	//Kommunikationsfel
	fbKommTof : tof; 
	fbKommTon : ton;
		
	fb_CSP : Tc3_BA.FB_BA_Chrct02;
	
	sIP: STRING(255);
	sPort: STRING(255);
	sModbusID: STRING(255);
	sModbusLoop: STRING(255);
	
	sTemp: STRING(255);
END_VAR

//General
	offset := 0;
//Sekvens	
	bSekvensFlagga := oaksGVL.aBModbusSekvens[iModbusLoop] = UINT_TO_INT(nUnitID);
//Modbus konfiguering
	sIP := CONCAT (SIPAddr, '');
	sPort := CONCAT ('<br>Port: ', UINT_TO_STRING(nTCPPort)); 								
	sModbusID := CONCAT('<br>ID: ', UINT_TO_STRING(nUnitID));
	sModbusLoop := CONCAT('<br>Loop: ', INT_TO_STRING(iModbusLoop));
	
	sTemp := sIP;
	sTemp := CONCAT(sTemp, sPort);
	sTemp := CONCAT(sTemp, sModbusID);
	sTemp := CONCAT(sTemp, sModbusLoop);
	
	PV10 := sTemp;

///////////////		
//READ
///////////////		
	
	//Read Holding 0-8
	FB_MBReadRegs_ArrHolding1(
	sIPAddr:= sIpAddr, 
	nTCPPort:= INT_TO_UINT(nTCPPort), 
	nUnitID:= INT_TO_BYTE(nUnitID), 
	nQuantity:= 9, 
	nMBAddr:= 0 + offset, 
	cbLength:= SIZEOF(ArrHolding1), 
	pDestAddr:= ADR(ArrHolding1), 
	bExecute:= bSekvensFlagga, 
	tTimeout:= T#3S, 
	bBusy=> , 
	bError=> , 
	nErrId=> , 
	cbRead=> );
	
		//Values
		wActSetpoint := ArrHolding1[0]; //0
		wModeOut := ArrHolding1[1]; //1
		//ArrHolding1[2]; //2
		//ArrHolding1[3]; //3
		//ArrHolding1[4]; //4
		wRelPos := ArrHolding1[5]; //5
		//ArrHolding1[6]; //6
		wAbsVolume := ArrHolding1[7]; //7
		//ArrHolding1[8]; //8
							
		//Absolute Volume flow
		//Converter from m2 to l/s
		iTemp := WORD_TO_UINT(wAbsVolume);
		rTemp := UINT_TO_REAL(iTemp);
		PV1 := rTemp;
	
		//Relative Position
		iTemp := WORD_TO_UINT(wRelPos);
		rTemp := UINT_TO_REAL(iTemp);
		OP := rTemp / 100;
		
		//Actual damper-mode
		PV5 := wModeOut;
						
	//Read Holding 100-108
	FB_MBReadRegs_ArrHolding2(
	sIPAddr:= sIpAddr, 
	nTCPPort:= INT_TO_UINT(nTCPPort), 
	nUnitID:= INT_TO_BYTE(nUnitID), 
	nQuantity:= 9, 
	nMBAddr:= 100 + offset, 
	cbLength:= SIZEOF(ArrHolding2), 
	pDestAddr:= ADR(ArrHolding2), 
	bExecute:= bSekvensFlagga, 
	tTimeout:= T#3S, 
	bBusy=> , 
	bError=> , 
	nErrId=> , 
	cbRead=> );
	
		//Tilldela värden
		//ArrHolding2[100]; //100
		//ArrHolding2[101]; //101
		//ArrHolding2[102]; //102
		//ArrHolding2[103]; //103
		//ArrHolding2[104]; //104
		wAlarm := ArrHolding2[105]; //105
		//ArrHolding2[106]; //106
		//ArrHolding2[107]; //107
		//ArrHolding2[108]; //108
		
	
	//Read Holding 120-122
	FB_MBReadRegs_ArrHolding3(
	sIPAddr:= sIpAddr, 
	nTCPPort:= INT_TO_UINT(nTCPPort), 
	nUnitID:= INT_TO_BYTE(nUnitID), 
	nQuantity:= 3, 
	nMBAddr:= 120 + offset, 
	cbLength:= SIZEOF(ArrHolding3), 
	pDestAddr:= ADR(ArrHolding3), 
	bExecute:= bSekvensFlagga, 
	tTimeout:= T#3S, 
	bBusy=> , 
	bError=> , 
	nErrId=> , 
	cbRead=> );
	
		
		wMinVolume := ArrHolding3[120]; //120
		wMaxVolume := ArrHolding3[121]; //121		
		//ArrHolding3[122]; //122		
			
		//Setpoint Min-volume
		iTemp := WORD_TO_UINT(wMinVolume);
		PV6 := UINT_TO_REAL(iTemp);
						
		//Setpoint Max-volume
		iTemp := WORD_TO_UINT(wMaxVolume);
		PV7 := UINT_TO_REAL(iTemp);
		
	//Calculated setpoint
		fb_CSP(
			rX:= WORD_TO_REAL(wActSetpoint) / 100, 
			rX01:= 0, 
			rX02:= 100, 
			rY01:= PV6, 
			rY02:= PV7, 
			bLmt:= TRUE, 
			rY=> CSP, 
			bErr=> , 
			sErrDescr=> );

		
///////////////		
//WRITE
///////////////	
				
//Setpoint
	
	rTemp := LIMIT (0, rSetpoint, 100);
	wTemp := frealtoword(rTemp, 100);
		
	IF wTemp <> wActSetpoint AND bSekvensFlagga THEN
		FB_MBWriteSingleReg_Setpoint.bExecute := TRUE;
	ELSE
		FB_MBWriteSingleReg_Setpoint.bExecute := FALSE;
	END_IF
	
	//Write Setpoint
	FB_MBWriteSingleReg_Setpoint(
	sIPAddr:= sIpAddr, 
	nTCPPort:= INT_TO_UINT(nTCPPort), 
	nUnitID:= INT_TO_BYTE(nUnitID), 
	nMBAddr:= 0 + offset, 
	nValue:= wTemp, 
	bExecute:= , 
	tTimeout:= T#3S, 
	bBusy=> , 
	bError=> , 
	nErrId=> );
	
//Override
	
	iTemp := INT_TO_WORD(iMode);	

	IF wModeOut <> iTemp AND bSekvensFlagga THEN 
		FB_MBWriteSingleReg_Mode.bExecute := TRUE;
	ELSE 
		FB_MBWriteSingleReg_Mode.bExecute := FALSE;
	END_IF
	
	//Write Mode
	FB_MBWriteSingleReg_Mode(
	sIPAddr:= sIpAddr, 
	nTCPPort:= INT_TO_UINT(nTCPPort), 
	nUnitID:= INT_TO_BYTE(nUnitID), 
	nMBAddr:= 1 + offset, 
	nValue:= UINT_TO_WORD(iMode), 
	bExecute:= , 
	tTimeout:= T#3S, 
	bBusy=> , 
	bError=> , 
	nErrId=> );

//Read/write

//Min		
	fbWriteHoldingDoubleControlledMin(
	sIPAddr:= sIPAddr, 
	nTCPPort:= nTCPPort, 
	nUnitID:= UINT_TO_BYTE(nUnitID) , 
	nMBAddr:= 120+offset,
	bExecute:= bSekvensFlagga, 
	rScale:=1 , 
	rWrite:= SP1, 
	bBusy=> , 
	bError=> );
//Max
	fbWriteHoldingDoubleControlledMax(
	sIPAddr:= sIPAddr, 
	nTCPPort:= nTCPPort, 
	nUnitID:= UINT_TO_BYTE(nUnitID) , 
	nMBAddr:= 121+offset, 
	bExecute:=bSekvensFlagga , 
	rScale:=1 , 
	rWrite:=SP2 , 
	bBusy=> , 
	bError=> );
	
//Communication error
	fbKommTof(IN:=FB_MBReadRegs_ArrHolding1.bError , PT:=T#20S , Q=> , ET=> );
	fbKommTon(IN:=fbKommTof.Q , PT:=T#20M , Q=> , ET=> );
	FAULT :=fbKommTon.Q;
		
//Write busy	
	oaksgvl.aBModbusBusyFlagga[iModbusLoop,nUnitID] := FB_MBReadRegs_Arrholding1.bBusy OR FB_MBReadRegs_Arrholding2.bBusy OR FB_MBReadRegs_Arrholding3.bBusy OR FB_MBWriteSingleReg_Setpoint.bBusy OR FB_MBWriteSingleReg_Mode.bBusy;

END_FUNCTION_BLOCK

// oaksModbusLibrary/Frico/fbFricoSirE
// Modbusblock för frico sir e fläktluftvärmare fungerar bra men går att vidareutveckla med fler register
FUNCTION_BLOCK fbFricoSirE
VAR_INPUT
	sIPAddr : STRING := ''; 
	nTCPPort : UINT;
	nUnitID : UINT;
	iModbusLoop : INT :=1; //Modbusslinga
	M AT %M*  : BOOL;  //Reset summalarm~wp:
END_VAR
VAR_OUTPUT 
	V AT %M*  : BOOL;//Driftindikering~wp:[trendoptions]i:14400, t:1
	PV AT %M*  : REAL;//Temperatur~wp:[unit]°C[format]0.0[trendoptions]i:300
	PV1 AT %M*  : REAL;//Fläkthastighet~wp:[unit]%[format]0[trendoptions]i:300
	VALVE_OP AT %M*  : REAL;//Ventilläge~wp:[unit]%[format]0[trendoptions]i:300
	AL AT %M*  : BOOL; //Summalarm~wp:[trendoptions]i:300
	PV8 AT %M* : STRING;//Modbus konfiguering~wp:
	FAULT AT %M* : BOOL;//Kommunikationsfel~wp:[trendoptions]i:300
END_VAR
VAR
	sIP: STRING(255);
	sPort: STRING(255);
	sModbusID: STRING(255);
	sModbusLoop: STRING(255);
	sTemp : STRING(255);	


	//Kommunikationsfel
	fbKommTof : tof; 
	fbKommTon : ton;

	bSekvensFlagga : BOOL;	

	fbWriteToggle01,fbReadToggle : fbToggle;
	bExecute1,bExecute11,bExecute12 : BOOL;
	fbTemperature: FB_MBReadRegs;
	wWord :  ARRAY [1..9] OF WORD;
	wDaySetpointConfirmed,wNightSetpointConfirmed : WORD;
	
	
	
	fbWriteNight: FB_MBWriteSingleReg;
	wDaySetpoint : WORD;
	fbWriteToggle011 : fbToggle;
	
	fbWriteDay: FB_MBWriteSingleReg;
	wNightSetpoint : WORD;
	fbWriteToggle012 : fbToggle;
	
	
	wResetConfirmed : WORD;
		iTemp : INT;
	fbResetConfirmed : FB_MBReadRegs;
	fbWriteReset: FB_MBWriteSingleReg;
END_VAR
VAR_INPUT PERSISTENT
	SP AT %M*  : REAL := 18;  //Inställt börvärde~wp:[unit]°C[format]0.0[trendoptions]i:300
END_VAR

//Modbus konfiguering
	sIP := CONCAT (SIPAddr, '');
	sPort := CONCAT ('<br>Port: ', UINT_TO_STRING(nTCPPort)); 								
	sModbusID := CONCAT('<br>ID: ', UINT_TO_STRING(nUnitID));
	sModbusLoop := CONCAT('<br>Loop: ', INT_TO_STRING(iModbusLoop));	

	sTemp := sIP;
	sTemp := CONCAT(sTemp, sPort);
	sTemp := CONCAT(sTemp, sModbusID);
	sTemp := CONCAT(sTemp, sModbusLoop);
	
	PV8 := sTemp;

//Sekvens	
	bSekvensFlagga := oaksGVL.aBModbusSekvens[iModbusLoop] = UINT_TO_INT(nUnitID);

	fbTemperature(
	sIPAddr:= sIPAddr, 
	nTCPPort:= nTCPPort, 
	nUnitID:= UINT_TO_BYTE(nUnitID), 
	nQuantity:= 9, 
	nMBAddr:= 0, 
	cbLength:= SIZEOF(wWord), 
	pDestAddr:=ADR(wWord) , 
	bExecute:=bSekvensFlagga , 
	tTimeout:= T#5S, 
	bBusy=> , 
	bError=> , 
	nErrId=> , 
	cbRead=> );

	PV := fSignedConverter(WORD_TO_REAL(wWord[1])) * 0.1;
	PV1 := WORD_TO_REAL(wWord[3]);
	VALVE_OP :=  WORD_TO_REAL(wWord[4]);
	
	V := PV1 > 0.0;
	
	
	wDaySetpointConfirmed := wWord[8];
	wNightSetpointConfirmed := wWord[9];
	
	IF mBHyst(rProcessValue :=SP ,rSetPoint:=REAL_TO_WORD(wDaySetpointConfirmed) ,rDevLimit:=0.25) THEN
		wDaySetpoint := REAL_TO_WORD(SP);
		bExecute11 := TRUE;
	ELSE
		bExecute11 := FALSE;
	END_IF;
	
	fbWriteToggle011(bStart:=bExecute11 , bOutput=> );

	fbWriteDay(
	sIPAddr:= sIpAddr, 
	nTCPPort:= INT_TO_UINT(nTCPPort), 
	nUnitID:= INT_TO_BYTE(nUnitID), 
	nMBAddr:= 7, 
	nValue:= wDaySetpoint, 
	bExecute:= fbWriteToggle011.bOutput AND bSekvensFlagga, 
	tTimeout:=T#5S , 
	bBusy=> , 
	bError=> , 
	nErrId=> );
	
	IF mBHyst(rProcessValue :=SP ,rSetPoint:=REAL_TO_WORD(wNightSetpointConfirmed) ,rDevLimit:=0.25) THEN
		wNightSetpoint := REAL_TO_WORD(SP);
		bExecute12 := TRUE;
	ELSE
		bExecute12 := FALSE;
	END_IF;
	
	fbWriteToggle012(bStart:=bExecute12 , bOutput=> );

	fbWriteNight(
	sIPAddr:= sIpAddr, 
	nTCPPort:= INT_TO_UINT(nTCPPort), 
	nUnitID:= INT_TO_BYTE(nUnitID), 
	nMBAddr:= 8, 
	nValue:= wNightSetpoint, 
	bExecute:= fbWriteToggle012.bOutput AND bSekvensFlagga, 
	tTimeout:=T#5S , 
	bBusy=> , 
	bError=> , 
	nErrId=> );
(**** RESET START ****)
	IF M AND  wResetConfirmed = 0 THEN
		bExecute1 := TRUE;
	ELSE
		M := FALSE;
		bExecute1 := FALSE;
	END_IF;
	
	fbWriteToggle01(bStart:=bExecute1 , bOutput=> );

	fbWriteReset(
	sIPAddr:= sIpAddr, 
	nTCPPort:= INT_TO_UINT(nTCPPort), 
	nUnitID:= INT_TO_BYTE(nUnitID), 
	nMBAddr:= 99, 
	nValue:= 1, 
	bExecute:= fbWriteToggle01.bOutput AND bSekvensFlagga, 
	tTimeout:=T#1S , 
	bBusy=> , 
	bError=> , 
	nErrId=> );
	
	fbResetConfirmed(
	sIPAddr:= sIpAddr, 
	nTCPPort:= INT_TO_UINT(nTCPPort), 
	nUnitID:= INT_TO_BYTE(nUnitID), 
	nQuantity:= 1, 
	nMBAddr:= 99, 
	cbLength:= SIZEOF(wResetConfirmed), 
	pDestAddr:= ADR(wResetConfirmed), 
	bExecute:= bSekvensFlagga, 
	tTimeout:= T#1S, 
	bBusy=> , 
	bError=> , 
	nErrId=> , 
	cbRead=> );
	(**** RESET SLUT ****)
	
	//Communication error
	fbKommTof(IN:=fbTemperature.bError , PT:=T#20S , Q=> , ET=> );
	fbKommTon(IN:=fbKommTof.Q , PT:=T#20M , Q=> , ET=> );
	FAULT :=fbKommTon.Q;
		
//Write busy	
	oaksgvl.aBModbusBusyFlagga[iModbusLoop,nUnitID] := fbResetConfirmed.bBusy OR fbWriteReset.bBusy OR fbWriteNight.bBusy OR fbWriteDay.bBusy OR fbTemperature.bBusy;

METHOD PRIVATE mBHyst : BOOL
VAR_INPUT
	rProcessValue : REAL;
	rSetPoint : REAL; 
	rDevLimit : REAL;
END_VAR
VAR
END_VAR
	IF rProcessValue > (rSetPoint + rDevLimit)  THEN
		mBHyst := TRUE;
	ELSIF rProcessValue < (rSetPoint - rDevLimit)  THEN
		mBHyst := TRUE;
	ELSE	
		mBHyst := FALSE;
	END_IF;
END_METHOD

END_FUNCTION_BLOCK

// oaksModbusLibrary/Frico/fbFricoSirEOvride
// Modbusblock för frico sir e fläktluftvärmare fungerar bra men går att vidareutveckla med fler register
//2023-01-20 v2 Johan Stenström, Lagt till skicka utetemp., start/stopp, växling dag/natt

FUNCTION_BLOCK fbFricoSirEOvride
VAR_INPUT
	sIPAddr : STRING := ''; 
	nTCPPort : UINT := 502;
	nUnitID : UINT;
	iModbusLoop : INT := 1; //Modbusslinga
	iOnOff AT %M* : INT := 1; //Extern styrning till/från~wp:
	PV6 AT %M* : INT := 1; //Dag/Natt styrning börvärde, Dag=1, Natt=0~wp:
	ACK AT %M* : BOOL;  //Reset summalarm~wp:
END_VAR
VAR_OUTPUT 
	V AT %M*  : BOOL;//Driftindikering~wp:[trendoptions]i:14400, t:1
	CMD AT %M* : BOOL ; //Manöver~wp:[trendoptions]i:14400, t:1
	ROOM_PV AT %M*  : REAL;//Temperatur~wp:[unit]°C[format]0.0[trendoptions]i:300
	ROOM_CSP AT %M*  : REAL;//Aktuellt börvärde~wp:[unit]°C[format]0.0[trendoptions]i:300
	PV1 AT %M*  : REAL;//Fläkthastighet~wp:[unit]%[format]0[trendoptions]i:300
	VALVE_OP AT %M*  : REAL;//Ventilläge~wp:[unit]%[format]0[trendoptions]i:300
	AL AT %M*  : BOOL; //Summalarm~wp:[alarmoptions]p:2
	AL8 AT %M* : BOOL; //Utsignal handställd~wp:[alarmoptions]p:3
	PV8 AT %M* : STRING;//Modbus konfiguering~wp:
	FAULT AT %M* : BOOL;//Kommunikationsfel~wp:[trendoptions]i:300
END_VAR
VAR
	sIP: STRING(255);
	sPort: STRING(255);
	sModbusID: STRING(255);
	sModbusLoop: STRING(255);
	sTemp : STRING(255);	
	offset : WORD;
	fbAlarm1 : fbAlarm; // Larm handställning
//Kommunikationsfel
	fbKommTof : tof; 
	fbKommTon : ton;

	bSekvensFlagga : BOOL;	

	fbWriteToggle01 : fbToggle;
	bExecute1 : BOOL; 
	fbTemperature : FB_MBReadRegs;
	wWord :  ARRAY [1..12] OF WORD;
	wWordAlarm :  ARRAY [1..33] OF WORD;
	rOutDoorTempPointValueConfirmed : REAL;
	wSystemOnOffConfirmed, wWeekProgramConfirmed : WORD;
	wDaySetpointConfirmed, wNightSetpointConfirmed : WORD;
//OutDoorTemp	
	fbWriteOutDoorTemp : FB_MBWriteSingleReg;
	wOutDoorTempPointValue : WORD;
//SystemOnOff
	fbSystemOnOff : FB_MBWriteSingleReg;
	wSystemOnOff : WORD;
//WeekProgram
	fbWeekProgram : FB_MBWriteSingleReg;
	wWeekProgram : WORD;
//Setpoint Day	
	fbWriteDay : FB_MBWriteSingleReg;
	wDaySetpoint : WORD;
//Setpoint Night	
	fbWriteNight : FB_MBWriteSingleReg;
	wNightSetpoint : WORD;
//Alarm	
	fbAlarm : FB_MBReadRegs;
	wResetConfirmed : WORD;
//	iTemp : INT;
	fbResetConfirmed : FB_MBReadRegs;
	fbWriteReset : FB_MBWriteSingleReg;
	bAlarm01 : BOOL;
	bAlarm02 : BOOL; 
	bAlarm03 : BOOL; 
	bAlarm04 : BOOL; 
	bAlarm06 : BOOL;
	bAlarm07 : BOOL;
	bAlarm08 : BOOL; 
	bAlarm10 : BOOL; 
	bAlarm12 : BOOL; 
	bAlarm14 : BOOL;
	bAlarm21 : BOOL;
	bAlarm29 : BOOL;
	bAlarm30 : BOOL; 
	bAlarm31 : BOOL; 
	bAlarm32 : BOOL; 
	bAlarm33 : BOOL;  
	
END_VAR
VAR_INPUT PERSISTENT
	PV5 AT %M* : REAL;//Utetemperatur~wp:[unit]°C[format]0.0
	DAY_SP AT %M*  : REAL := 18;  //Börvärde dag~wp:[unit]°C[format]0.0[trendoptions]i:300
	NIGHT_SP AT %M*  : REAL := 16;  //Börvärde natt~wp:[unit]°C[format]0.0[trendoptions]i:300
	M AT %M* : BOOL; //Handställning~wp:
	MCMD AT %M* : BOOL; //Styrsignal handställning~wp:
END_VAR

//General
	offset := 0;
	fbAlarm1(bInput:=M, tAlarmDelay:= , bAutoReset:=TRUE , bAlarmOutput=>AL8 );
//Sekvens	
	bSekvensFlagga := oaksGVL.aBModbusSekvens[iModbusLoop] = UINT_TO_INT(nUnitID);
//Modbus konfiguering
	sIP := CONCAT (SIPAddr, '');
	sPort := CONCAT ('<br>Port: ', UINT_TO_STRING(nTCPPort)); 								
	sModbusID := CONCAT('<br>ID: ', UINT_TO_STRING(nUnitID));
	sModbusLoop := CONCAT('<br>Loop: ', INT_TO_STRING(iModbusLoop));	

	sTemp := sIP;
	sTemp := CONCAT(sTemp, sPort);
	sTemp := CONCAT(sTemp, sModbusID);
	sTemp := CONCAT(sTemp, sModbusLoop);
	
	PV8 := sTemp;
	
	IF PV6 > 0 THEN
		ROOM_CSP := DAY_SP;
	ELSE
		ROOM_CSP := NIGHT_SP;
	END_IF;

	fbTemperature(
	sIPAddr:= sIPAddr, 
	nTCPPort:= (nTCPPort), 
	nUnitID:= UINT_TO_BYTE(nUnitID), 
	nQuantity:= 10, 
	nMBAddr:= 0 + offset,
	cbLength:= SIZEOF(wWord), 
	pDestAddr:= ADR(wWord), 
	bExecute:= bSekvensFlagga, 
	tTimeout:= T#5S, 
	bBusy=> , 
	bError=> , 
	nErrId=> , 
	cbRead=> );

	ROOM_PV := fSignedConverter(WORD_TO_REAL(wWord[1])) * 0.1;
	rOutDoorTempPointValueConfirmed := fSignedConverter(WORD_TO_REAL(wWord[2]));
	PV1 := WORD_TO_REAL(wWord[3]);
	VALVE_OP :=  WORD_TO_REAL(wWord[4]);
	
	V := PV1 > 0.0;
	CMD := PV1 > 0.0;
	
	wSystemOnOffConfirmed := wWord[6];
	wWeekProgramConfirmed := wWord[7];
	wDaySetpointConfirmed := wWord[8];
	wNightSetpointConfirmed := wWord[9];
	
//OutDoorTemp	
	wOutDoorTempPointValue := fRealToWord(rReal:=PV5 , uiFaktor:= 10);
	
	fbWriteOutDoorTemp(
	sIPAddr:= sIpAddr, 
	nTCPPort:= INT_TO_UINT(nTCPPort), 
	nUnitID:= INT_TO_BYTE(nUnitID), 
	nMBAddr:= 1 + offset,
	nValue:= wOutDoorTempPointValue,
	bExecute:= bSekvensFlagga,
	tTimeout:=T#5S , 
	bBusy=> , 
	bError=> , 
	nErrId=> );	

//SystemOnOff	
	wSystemOnOff := INT_TO_WORD(iOnOff);
	
	IF M THEN
		IF (M AND MCMD) THEN
			wSystemOnOff := INT_TO_WORD(1);
		ELSE
			wSystemOnOff := INT_TO_WORD(0);
		END_IF
	ELSE
		wSystemOnOff := INT_TO_WORD(iOnOff);
	END_IF
	
	fbSystemOnOff(
	sIPAddr:= sIpAddr, 
	nTCPPort:= INT_TO_UINT(nTCPPort), 
	nUnitID:= INT_TO_BYTE(nUnitID), 
	nMBAddr:= 5 + offset, 
	nValue:= wSystemOnOff, 
	bExecute:= bSekvensFlagga,
	tTimeout:=T#5S , 
	bBusy=> , 
	bError=> , 
	nErrId=> );		
	
//WeekProgram
	IF PV6 > 0 THEN
		wWeekProgram := INT_TO_WORD(1);
	ELSE
		wWeekProgram := INT_TO_WORD(2);
	END_IF
	
	fbWeekProgram(
	sIPAddr:= sIpAddr, 
	nTCPPort:= INT_TO_UINT(nTCPPort), 
	nUnitID:= INT_TO_BYTE(nUnitID), 
	nMBAddr:= 6 + offset,
	nValue:= wWeekProgram, 
	bExecute:= bSekvensFlagga,
	tTimeout:=T#5S , 
	bBusy=> , 
	bError=> , 
	nErrId=> );		
	
//DaySetpoint
	wDaySetpoint := REAL_TO_WORD(DAY_SP);	

	fbWriteDay(
	sIPAddr:= sIpAddr, 
	nTCPPort:= INT_TO_UINT(nTCPPort), 
	nUnitID:= INT_TO_BYTE(nUnitID), 
	nMBAddr:= 7 + offset, 
	nValue:= wDaySetpoint, 
	bExecute:= bSekvensFlagga,
	tTimeout:=T#5S , 
	bBusy=> , 
	bError=> , 
	nErrId=> );
	
//WriteNight
	wNightSetpoint := REAL_TO_WORD(NIGHT_SP);

	fbWriteNight(
	sIPAddr:= sIpAddr, 
	nTCPPort:= INT_TO_UINT(nTCPPort), 
	nUnitID:= INT_TO_BYTE(nUnitID), 
	nMBAddr:= 8 + offset, 
	nValue:= wNightSetpoint, 
	bExecute:= bSekvensFlagga,
	tTimeout:=T#5S , 
	bBusy=> , 
	bError=> , 
	nErrId=> );
	
(**** ALARM ****)	
	bSekvensFlagga := oaksGVL.aBModbusSekvens[iModbusLoop] = UINT_TO_INT(nUnitID);

	fbAlarm(
	sIPAddr:= sIPAddr, 
	nTCPPort:= nTCPPort, 
	nUnitID:= UINT_TO_BYTE(nUnitID), 
	nQuantity:= 33, 
	nMBAddr:= 100 + offset, 
	cbLength:= SIZEOF(wWordAlarm), 
	pDestAddr:=ADR(wWordAlarm) , 
	bExecute:=bSekvensFlagga , 
	tTimeout:= T#5S, 
	bBusy=> , 
	bError=> , 
	nErrId=> , 
	cbRead=> );

	bAlarm01 := WORD_TO_BOOL(wWordAlarm[1]);
	bAlarm02 := WORD_TO_BOOL(wWordAlarm[2]);
	bAlarm03 := WORD_TO_BOOL(wWordAlarm[3]);
	bAlarm04 :=  WORD_TO_BOOL(wWordAlarm[4]);	
	bAlarm06 :=  WORD_TO_BOOL(wWordAlarm[6]);
	bAlarm07 :=  WORD_TO_BOOL(wWordAlarm[7]);
	bAlarm08 :=  WORD_TO_BOOL(wWordAlarm[8]);
	bAlarm10 :=  WORD_TO_BOOL(wWordAlarm[10]);
	bAlarm12 :=  WORD_TO_BOOL(wWordAlarm[12]);
	bAlarm14 :=  WORD_TO_BOOL(wWordAlarm[14]);
	bAlarm21 :=  WORD_TO_BOOL(wWordAlarm[21]);
	bAlarm29 :=  WORD_TO_BOOL(wWordAlarm[29]);
	bAlarm30 :=  WORD_TO_BOOL(wWordAlarm[30]);
	bAlarm31 :=  WORD_TO_BOOL(wWordAlarm[31]);
	bAlarm32 :=  WORD_TO_BOOL(wWordAlarm[32]);
	bAlarm33 :=  WORD_TO_BOOL(wWordAlarm[33]);
	
	IF bAlarm01 OR bAlarm02 OR bAlarm03 OR bAlarm04 OR bAlarm06 OR	bAlarm07 OR
		bAlarm08 OR bAlarm10 OR	bAlarm12 OR bAlarm14 OR bAlarm21 OR	bAlarm29 OR
		bAlarm30 OR bAlarm31 OR	bAlarm32 OR bAlarm33 = TRUE THEN
		AL := TRUE;
	ELSE
		AL := FALSE;
	END_IF;	
	
(**** RESET START ****)
	IF ACK AND  wResetConfirmed = 0 THEN
		bExecute1 := TRUE;
	ELSE
		ACK := FALSE;
		bExecute1 := FALSE;
	END_IF;
	
	fbWriteToggle01(bStart:=bExecute1 , bOutput=> );

	fbWriteReset(
	sIPAddr:= sIpAddr, 
	nTCPPort:= INT_TO_UINT(nTCPPort), 
	nUnitID:= INT_TO_BYTE(nUnitID), 
	nMBAddr:= 99 + offset, 
	nValue:= 1, 
	bExecute:= fbWriteToggle01.bOutput AND bSekvensFlagga, 
	tTimeout:=T#1S , 
	bBusy=> , 
	bError=> , 
	nErrId=> );
	
	fbResetConfirmed(
	sIPAddr:= sIpAddr, 
	nTCPPort:= INT_TO_UINT(nTCPPort), 
	nUnitID:= INT_TO_BYTE(nUnitID), 
	nQuantity:= 1, 
	nMBAddr:= 99, 
	cbLength:= SIZEOF(wResetConfirmed), 
	pDestAddr:= ADR(wResetConfirmed), 
	bExecute:= bSekvensFlagga, 
	tTimeout:= T#1S, 
	bBusy=> , 
	bError=> , 
	nErrId=> , 
	cbRead=> );
	(**** RESET SLUT ****)
	
//Communication error
	fbKommTof(IN:=fbTemperature.bError , PT:=T#10S , Q=> , ET=> );
	fbKommTon(IN:=fbKommTof.Q , PT:=T#20M , Q=> , ET=> );
	FAULT :=fbKommTon.Q;
		
//Write busy	
	oaksgvl.aBModbusBusyFlagga[iModbusLoop,nUnitID] := fbResetConfirmed.bBusy OR fbWriteReset.bBusy OR fbWriteNight.bBusy OR fbWriteDay.bBusy OR fbWeekProgram.bBusy OR fbSystemOnOff.bBusy OR fbWriteOutDoorTemp.bBusy OR fbTemperature.bBusy;

METHOD PRIVATE mBHyst : BOOL
VAR_INPUT
	rProcessValue : REAL;
	rSetPoint : REAL; 
	rDevLimit : REAL;
END_VAR
VAR
END_VAR
	IF rProcessValue > (rSetPoint + rDevLimit)  THEN
		mBHyst := TRUE;
	ELSIF rProcessValue < (rSetPoint - rDevLimit)  THEN
		mBHyst := TRUE;
	ELSE	
		mBHyst := FALSE;
	END_IF;
END_METHOD

END_FUNCTION_BLOCK

// oaksModbusLibrary/Grundfil/fbGrundfil
//OAKS AB
//2020-05-12
//Grundfil för modbusblock
FUNCTION_BLOCK fbGrundfil
VAR_INPUT
	sIPAddr : STRING := ''; 
	nTCPPort : UINT;
	nUnitID : UINT :=1;
	iModbusLoop : INT :=1; //Modbusslinga
			
END_VAR
VAR_OUTPUT
		
	PV8 AT %M* : STRING;//Modbus konfiguering~wp:
	FAULT AT %M* : BOOL;//Kommunikationsfel~wp:
	
END_VAR
VAR
	offset : WORD;
	rTemp : REAL;
	iTemp : UINT;
	bSekvensFlagga : BOOL;
			
	FB_MBReadRegs_ArrHolding1: FB_MBReadRegs;
	ArrHolding1 : ARRAY [0..10] OF WORD; //Holding
		
	//Kommunikationsfel
	fbKommTof : tof; 
	fbKommTon : fbAlarm;
	
	sIP: STRING(255);
	sPort: STRING(255);
	sModbusID: STRING(255);
	sModbusLoop: STRING(255);
	sTemp : STRING(255);
	
	
END_VAR

//General
	offset := 0;
//Sekvens	
	bSekvensFlagga := oaksGVL.aBModbusSekvens[iModbusLoop] = UINT_TO_INT(nUnitID);
//Modbus konfiguering
	sIP := CONCAT (SIPAddr, '');
	sPort := CONCAT ('<br>Port: ', UINT_TO_STRING(nTCPPort)); 								
	sModbusID := CONCAT('<br>ID: ', UINT_TO_STRING(nUnitID));
	sModbusLoop := CONCAT('<br>Loop: ', INT_TO_STRING(iModbusLoop));	

	sTemp := sIP;
	sTemp := CONCAT(sTemp, sPort);
	sTemp := CONCAT(sTemp, sModbusID);
	sTemp := CONCAT(sTemp, sModbusLoop);
	
	PV8 := sTemp;

///////////////		
//READ
///////////////		
	
	//Read Holding 0-10
	FB_MBReadRegs_ArrHolding1(
	sIPAddr:= sIpAddr, 
	nTCPPort:= INT_TO_UINT(nTCPPort), 
	nUnitID:= INT_TO_BYTE(nUnitID), 
	nQuantity:= 1, 
	nMBAddr:= 0 + offset, 
	cbLength:= SIZEOF(ArrHolding1), 
	pDestAddr:= ADR(ArrHolding1), 
	bExecute:= bSekvensFlagga, 
	tTimeout:= T#3S, 
	bBusy=> , 
	bError=> , 
	nErrId=> , 
	cbRead=> );
	
		//Values
		//ArrHolding1[0]; //0
		//ArrHolding1[1]; //1
		//ArrHolding1[2]; //2
		//ArrHolding1[3]; //3
		//ArrHolding1[4]; //4
		//ArrHolding1[5]; //5
		//ArrHolding1[6]; //6
		//ArrHolding1[7]; //7
		//ArrHolding1[8]; //8
		//ArrHolding1[9]; //9
		//ArrHolding1[10]; //10
		
	
//Communication error
	fbKommTof(IN:=FB_MBReadRegs_ArrHolding1.bError , PT:=T#20S , Q=> , ET=> );
	fbKommTon(bInput:=fbKommTof.Q , tAlarmDelay:=T#20M , bAutoReset:= , bAlarmOutput=> );
	FAULT :=fbKommTon.bAlarmOutput;
		
//Write busy	
	oaksgvl.aBModbusBusyFlagga[iModbusLoop,nUnitID] := FB_MBReadRegs_Arrholding1.bBusy;

END_FUNCTION_BLOCK

// oaksModbusLibrary/Grundfos/fbGrundfosCIM
//Funktionsblock för kommunikation mot kom.modul Grundfos CIM200/500 (via ModbusTCP-gateway). Skriv larmreset, läsning av div. värden
//Robert H Oaks AB 
//22-03-16

//V 1.0	Testad

//OBS! Ej anpassad för Modbus-sekvens i oaks-standard, bör åtgärdas!!

(*

00101.2		ResetAlarm

00201.6		Rotation
00201.9		OnOff
00201.10	Fault
00201.11	Warning
00201.12	ForcedToLocal

00202		ProcessFeedback 		0.00 %
00205		AlarmCode
00206		WarningCode
00208		DriveState

00301		Head					0.001 bar
00302		VolumeFlow				0.1 m3/h
00303		RelativePerformance		0.01 %
00304		Speed					1 rpm
00305		Frequency				0.1 Hz
00309		MotorCurrent			0.1 A
00310		DCLinkVoltage			0.1 V
00311		MotorVoltage			0.1 V
00312-313	PowerHI/LO				1 W
00318		PowerElectronicTemp		0.01 K
00319		MotorTemp				0.01 K
00321		ElectronicTemp			0.01 K
00322		PumpLiquidTemp			0.01 K
00327-328	OperationTimeHI/LO		1 hour
00329-330	TotalPoweredTimeHi/LO	1 hour
00332-333	EnergyHI/LO				1 kWh
00334-335	NumberOfStartsHI/LO		1 start


*)



FUNCTION_BLOCK fbGrundfosCIM
VAR_INPUT
	sIPAddr 		: STRING; 			//Ip-adress till ModbusTCP-gateway
	nMBTCPPort		: UINT := 502;		//ModbusTCP-port
	nUnitID			: UINT := 1;		//Enhetsadress
	tInterval		: TIME := T#3S;		//Kommunikationsintervall
	tTimeout		: TIME := T#2S;		//Timeout
	CMD AT %M*		: BOOL;				//Larmreset ~wp: 
END_VAR

VAR_OUTPUT
	V1		AT %M*		: BOOL;				//Motor i drift~wp:[trendoptions]i:14400, t:1
	V2		AT %M*		: BOOL;				//Pump aktiverad~wp:[trendoptions]i:14400, t:1		
	FAULT	AT %M*		: BOOL;				//Fellarm från pumpstyrning~wp:[alarmoptions]p:2
	AL1		AT %M*		: BOOL;				//Varning från pumpstyrning~wp:[alarmoptions]p:2
	AL2		AT %M*		: BOOL;				//Pump i lokal drift~wp:[alarmoptions]p:3
	AL8		AT %M*		: BOOL;				//Kommunikationsfel styrenhet pump~wp:[alarmoptions]p:3
	
	PV1		AT %M* 		: STRING := '';		//Driftläge~wp:
	PV2		AT %M* 		: REAL; 			//Faktisk driftnivå~wp:[unit]%[format]0[trendoptions]i:300
	//PV3		AT %M* 		: REAL; 			//Systemtryck~wp:[unit]kPa[format]0.0[trendoptions]i:300
	//PV4		AT %M* 		: REAL; 			//Flöde~wp:[unit]m3/h[format]0.0[trendoptions]i:300
	PV5		AT %M* 		: REAL; 			//Pumphastighet~wp:[unit]rpm[format]0[trendoptions]i:300
	PV6		AT %M* 		: REAL; 			//Motorfrekvens~wp:[unit]Hz[format]0.0[trendoptions]i:300
	PV7		AT %M* 		: REAL; 			//Motorström~wp:[unit]A[format]0.0[trendoptions]i:300
	PV8		AT %M* 		: REAL; 			//DC-spänning FO~wp:[unit]V[format]0.0[trendoptions]i:300
	PV9		AT %M* 		: REAL; 			//Motorspänning~wp:[unit]V[format]0.0[trendoptions]i:300
	PV10	AT %M* 		: REAL; 			//Motoreffekt~wp:[unit]kW[format]0.00[trendoptions]i:300
	PV11	AT %M* 		: UDINT; 			//Drifttid pump~wp:[unit]h[format]0[trendoptions]i:300
	PV12	AT %M* 		: UDINT; 			//Drifttid elektronik~wp:[unit]h[format]0[trendoptions]i:300
	PV13	AT %M* 		: UDINT; 			//Elförbruknig pump~wp:[unit]kWh[format]0[trendoptions]i:300
	PV14	AT %M* 		: UDINT; 			//Antal starter~wp:[unit]st[format]0[trendoptions]i:14400, t:1
	PV15	AT %M* 		: UINT; 			//Felkod styrenhet~wp:[format]0[trendoptions]i:14400, t:1
	PV16	AT %M* 		: UINT; 			//Varningskod styrenhet~wp:[format]0[trendoptions]i:14400, t:1
END_VAR

VAR
	bRun			: BOOL;	
	fbRunTON		: TON;
	fbRunTRIG		: R_TRIG;
	
	bDidRead		: BOOL;

	fbR00101		: FB_MBReadRegs;
	fbW00101		: FB_MBWriteSingleReg;
	
	fbR00201		: FB_MBReadRegs;
	fbR00202		: FB_MBReadRegs;
	fbR00205		: FB_MBReadRegs;
	fbR00206		: FB_MBReadRegs;
	fbR00208		: FB_MBReadRegs;
	fbR00301		: FB_MBReadRegs;
	fbR00302		: FB_MBReadRegs;
	fbR00304		: FB_MBReadRegs;
	fbR00305		: FB_MBReadRegs;
	fbR00309		: FB_MBReadRegs;
	fbR00310		: FB_MBReadRegs;
	fbR00311		: FB_MBReadRegs;
	fbR00312_313	: FB_MBReadRegs;
	fbR00327_328	: FB_MBReadRegs;
	fbR00329_330	: FB_MBReadRegs;
	fbR00332_333	: FB_MBReadRegs;
	fbR00334_335	: FB_MBReadRegs;
	
	wR00101			: WORD;
	wR00201			: WORD;
	wR00202			: WORD;
	wR00205			: WORD;
	wR00206			: WORD;
	wR00208			: WORD;
	wR00301			: WORD;
	wR00302			: WORD;
	wR00304			: WORD;
	wR00305			: WORD;
	wR00309			: WORD;
	wR00310			: WORD;
	wR00311			: WORD;
	uR00312_313		: WORD2_TO_UDINT;
	uR00327_328		: WORD2_TO_UDINT;
	uR00329_330		: WORD2_TO_UDINT;
	uR00332_333		: WORD2_TO_UDINT;
	uR00334_335		: WORD2_TO_UDINT;
	
	fbErrorTOF		: TOF;
	fbErrorTON		: TON;
	
END_VAR

fbRunTON(IN := NOT bRun, PT := tInterval);
fbRunTRIG(CLK := fbRunTON.Q, Q => bRun);


//00101	Pump control register block		Endast larmreset. Läs in ord, då larmreset sätts från Webport skrivs ord tillbaks lika läsning med bit 2 hög	
IF CMD AND bRun THEN
	
	IF NOT bDidRead THEN
		fbR00101(sIPAddr := sIPAddr, nTCPPort := nMBTCPPort, nUnitID := UINT_TO_BYTE(nUnitID), nQuantity := 1, bExecute := bRun, tTimeout := tTimeout,   
			nMBAddr 	:= 100,
			cbLength	:= SIZEOF(wR00101),
			pDestAddr	:= ADR(wR00101));
			
		bDidRead := TRUE;
	ELSE
		IF NOT (fbR00101.bBusy OR fbR00101.bError) THEN
		
			wR00101.2 := TRUE;
		
			fbW00101(sIPAddr := sIPAddr, nTCPPort := nMBTCPPort, nUnitID := UINT_TO_BYTE(nUnitID), tTimeout := tTimeout,
				bExecute 	:= bRun,   
				nMBAddr 	:= 100,
				nValue		:= wR00101);
				
			bDidRead	:= FALSE;
			CMD 		:= FALSE;
		END_IF;
	END_IF;			
	
END_IF;

	
//00201	Pump status register block	
fbR00201(sIPAddr := sIPAddr, nTCPPort := nMBTCPPort, nUnitID := UINT_TO_BYTE(nUnitID), nQuantity := 1, bExecute := bRun, tTimeout := tTimeout,   
	nMBAddr 	:= 200,
	cbLength	:= SIZEOF(wR00201),
	pDestAddr	:= ADR(wR00201));
	V1		:= wR00201.6;
	V2		:= wR00201.9;
	FAULT	:= wR00201.10;
	AL1		:= wR00201.11;
	AL2		:= wR00201.12;
	
//00202	Process Feedback	
fbR00202(sIPAddr := sIPAddr, nTCPPort := nMBTCPPort, nUnitID := UINT_TO_BYTE(nUnitID), nQuantity := 1, bExecute := bRun, tTimeout := tTimeout,   
	nMBAddr 	:= 201,
	cbLength	:= SIZEOF(wR00202),
	pDestAddr	:= ADR(wR00202));
	PV2	:= wR00202 / 100;
	
//00205	Alarm Code	
fbR00205(sIPAddr := sIPAddr, nTCPPort := nMBTCPPort, nUnitID := UINT_TO_BYTE(nUnitID), nQuantity := 1, bExecute := bRun, tTimeout := tTimeout,   
	nMBAddr 	:= 204,
	cbLength	:= SIZEOF(wR00205),
	pDestAddr	:= ADR(wR00205));
	PV15		:= wR00205;

//00206	Warning Code	
fbR00206(sIPAddr := sIPAddr, nTCPPort := nMBTCPPort, nUnitID := UINT_TO_BYTE(nUnitID), nQuantity := 1, bExecute := bRun, tTimeout := tTimeout,   
	nMBAddr 	:= 205,
	cbLength	:= SIZEOF(wR00206),
	pDestAddr	:= ADR(wR00206));
	PV16		:= wR00206;
	
//00208	Drive State	
fbR00208(sIPAddr := sIPAddr, nTCPPort := nMBTCPPort, nUnitID := UINT_TO_BYTE(nUnitID), nQuantity := 1, bExecute := bRun, tTimeout := tTimeout,   
	nMBAddr 	:= 207,
	cbLength	:= SIZEOF(wR00208),
	pDestAddr	:= ADR(wR00208));
	
	CASE wR00208 OF 
		0:
		PV1	:= 'Stoppad';
		1:
		PV1	:= 'Rampar upp';
		2:
		PV1	:= 'Rampar ner';
		3:
		PV1	:= 'Stabil drift';
		5:
		PV1	:= 'Upprampning stopp';
		6:
		PV1	:= 'Nedrampning stopp';
		7:
		PV1	:= 'Flygande start';
	END_CASE;

//00301	Head
fbR00301(sIPAddr := sIPAddr, nTCPPort := nMBTCPPort, nUnitID := UINT_TO_BYTE(nUnitID), nQuantity := 1, bExecute := bRun, tTimeout := tTimeout,   
	nMBAddr 	:= 300,
	cbLength	:= SIZEOF(wR00301),
	pDestAddr	:= ADR(wR00301));
	//PV3			:= INT_TO_REAL(WORD_TO_INT(wR00301)) / 1000;
	
//00302	Volume flow
fbR00302(sIPAddr := sIPAddr, nTCPPort := nMBTCPPort, nUnitID := UINT_TO_BYTE(nUnitID), nQuantity := 1, bExecute := bRun, tTimeout := tTimeout,   
	nMBAddr 	:= 301,
	cbLength	:= SIZEOF(wR00302),
	pDestAddr	:= ADR(wR00302));
	//PV4			:= INT_TO_REAL(WORD_TO_INT(wR00302)) / 10;
	
//00304	Speed
fbR00304(sIPAddr := sIPAddr, nTCPPort := nMBTCPPort, nUnitID := UINT_TO_BYTE(nUnitID), nQuantity := 1, bExecute := bRun, tTimeout := tTimeout,   
	nMBAddr 	:= 303,
	cbLength	:= SIZEOF(wR00304),
	pDestAddr	:= ADR(wR00304));
	PV5			:= wR00304;
	
//00305	Frequency
fbR00305(sIPAddr := sIPAddr, nTCPPort := nMBTCPPort, nUnitID := UINT_TO_BYTE(nUnitID), nQuantity := 1, bExecute := bRun, tTimeout := tTimeout,   
	nMBAddr 	:= 304,
	cbLength	:= SIZEOF(wR00305),
	pDestAddr	:= ADR(wR00305));
	PV6			:= INT_TO_REAL(WORD_TO_INT(wR00305)) / 10;
	
//00309	Motor Current
fbR00309(sIPAddr := sIPAddr, nTCPPort := nMBTCPPort, nUnitID := UINT_TO_BYTE(nUnitID), nQuantity := 1, bExecute := bRun, tTimeout := tTimeout,   
	nMBAddr 	:= 308,
	cbLength	:= SIZEOF(wR00309),
	pDestAddr	:= ADR(wR00309));
	PV7			:= INT_TO_REAL(WORD_TO_INT(wR00309)) / 10;
	
//00310	DC Link Voltage
fbR00310(sIPAddr := sIPAddr, nTCPPort := nMBTCPPort, nUnitID := UINT_TO_BYTE(nUnitID), nQuantity := 1, bExecute := bRun, tTimeout := tTimeout,   
	nMBAddr 	:= 309,
	cbLength	:= SIZEOF(wR00310),
	pDestAddr	:= ADR(wR00310));
	PV8			:= INT_TO_REAL(WORD_TO_INT(wR00310)) / 10;
	
//00311	Motor Voltage
fbR00311(sIPAddr := sIPAddr, nTCPPort := nMBTCPPort, nUnitID := UINT_TO_BYTE(nUnitID), nQuantity := 1, bExecute := bRun, tTimeout := tTimeout,   
	nMBAddr 	:= 310,
	cbLength	:= SIZEOF(wR00311),
	pDestAddr	:= ADR(wR00311));
	PV9			:= INT_TO_REAL(WORD_TO_INT(wR00311)) / 10;
	
//00312-313	Power
fbR00312_313(sIPAddr := sIPAddr, nTCPPort := nMBTCPPort, nUnitID := UINT_TO_BYTE(nUnitID), bExecute := bRun, tTimeout := tTimeout,
	nQuantity 	:= 2,   
	nMBAddr 	:= 311,
	cbLength	:= SIZEOF(uR00312_313.aWdata),
	pDestAddr	:= ADR(uR00312_313.aWdata));
	PV10		:= DINT_TO_REAL(ROR(uR00312_313.ulCombined, 16)) / 1000;
	
//00327-328	Operation Time
fbR00327_328(sIPAddr := sIPAddr, nTCPPort := nMBTCPPort, nUnitID := UINT_TO_BYTE(nUnitID), bExecute := bRun, tTimeout := tTimeout,
	nQuantity 	:= 2,   
	nMBAddr 	:= 326,
	cbLength	:= SIZEOF(uR00327_328.aWdata),
	pDestAddr	:= ADR(uR00327_328.aWdata));
	
	IF (uR00327_328.aWdata[0] = 65535) AND (uR00327_328.aWdata[1] = 65535) THEN
		PV11	:= 0;
	ELSE
		PV11	:= ROR(uR00327_328.ulCombined, 16);
	END_IF
	
//00329-330	Total Powered Time
fbR00329_330(sIPAddr := sIPAddr, nTCPPort := nMBTCPPort, nUnitID := UINT_TO_BYTE(nUnitID), bExecute := bRun, tTimeout := tTimeout,
	nQuantity 	:= 2,   
	nMBAddr 	:= 328,
	cbLength	:= SIZEOF(uR00329_330.aWdata),
	pDestAddr	:= ADR(uR00329_330.aWdata));
	
	IF (uR00329_330.aWdata[0] = 65535) AND (uR00329_330.aWdata[1] = 65535) THEN
		PV12	:= 0;
	ELSE
		PV12	:= ROR(uR00329_330.ulCombined, 16);
	END_IF	
	
//00332-333	Energy
fbR00332_333(sIPAddr := sIPAddr, nTCPPort := nMBTCPPort, nUnitID := UINT_TO_BYTE(nUnitID), bExecute := bRun, tTimeout := tTimeout,
	nQuantity 	:= 2,   
	nMBAddr 	:= 331,
	cbLength	:= SIZEOF(uR00332_333.aWdata),
	pDestAddr	:= ADR(uR00332_333.aWdata));
	
	IF (uR00332_333.aWdata[0] = 65535) AND (uR00332_333.aWdata[1] = 65535) THEN
		PV13	:= 0;
	ELSE
		PV13	:= ROR(uR00332_333.ulCombined, 16);
	END_IF;
	
//00334-335	Number Of Starts
fbR00334_335(sIPAddr := sIPAddr, nTCPPort := nMBTCPPort, nUnitID := UINT_TO_BYTE(nUnitID), bExecute := bRun, tTimeout := tTimeout,
	nQuantity 	:= 2,   
	nMBAddr 	:= 333,
	cbLength	:= SIZEOF(uR00334_335.aWdata),
	pDestAddr	:= ADR(uR00334_335.aWdata));
	
	IF (uR00334_335.aWdata[0] = 65535) AND (uR00334_335.aWdata[1] = 65535) THEN
		PV14	:= 0;
	ELSE
		PV14	:= ROR(uR00334_335.ulCombined, 16);
	END_IF;
	
//Kom.fel modbus
fbErrorTOF(IN := fbR00101.bError, PT := T#30S);
fbErrorTON(IN := fbErrorTOF.Q, PT := T#120S, Q => AL8);

END_FUNCTION_BLOCK

// oaksModbusLibrary/Grundfos/fbGrundfosModbusMagna
//OAKS AB
//2020-05-12
//Grundfil för modbusblock
FUNCTION_BLOCK fbGrundfosModbusMagna
VAR_INPUT
	sIPAddr : STRING := ''; 
	nTCPPort : UINT;
	nUnitID : BYTE :=1;
	iModbusLoop : INT :=1; //Modbusslinga
	
END_VAR
VAR_OUTPUT
	PV8 AT %M* : STRING;//Modbus konfiguering~wp:
	FAULT AT %M* : BOOL;//Kommunikationsfel~wp:
	V AT %M* : BOOL; //Driftindikering~wp:[trendoptions]i:14400, t:1
	AL AT %M* : BOOL; //Fault error pump~wp:
	AL1 AT %M* : BOOL; //Warning error pump~wp:[alarmoptions]p:3
	AL2 AT %M* : BOOL; //Pump hand set~wp:[alarmoptions]p:3
	PV AT %M* :	REAL; //Energi~wp:[unit]kWh[format]0.0[trendoptions]i:300
	PV1 AT %M* :	REAL; //Effekt~wp:[unit]W[format]0[trendoptions]i:300
(* value array *) 
	PV2 AT %M* : REAL; //Tryck~wp:[unit]kPa[format]0.0[trendoptions]i:300
	PV3 AT %M* : REAL; //Flöde~wp:[unit]m3/h[format]0.0[trendoptions]i:300
	PV4 AT %M* : REAL; //Varvtal~wp:[unit]rpm[format]0[trendoptions]i:300
	PV5 AT %M* : REAL; //Frekvens~wp:[unit]Hz[format]0[trendoptions]i:300
	PV6 AT %M* : REAL; //Ström~wp:[unit]A[format]0.0[trendoptions]i:300
	PV7 AT %M* : REAL; //Drifttid~wp:[unit]timmar[format]0[trendoptions]i:300
END_VAR
VAR
	offset : WORD;
	rTemp : REAL;
	iTemp : UINT;
	bSekvensFlagga : BOOL;
	iTemp2 : UINT;	
	//Kommunikationsfel
	fbKommTof : tof; 
	fbKommTon : fbAlarm;
	
	sIP: STRING(255);
	sPort: STRING(255);
	sModbusID: STRING(255);
	sModbusLoop: STRING(255);
	sTemp : STRING(255);
	

	iBitHolder1,iBitHolder2,iBitHolder3 : WORD;
	
	fbReadEnergy	: FB_MBReadRegs;
	
	
	fbStatusBits : FB_MBReadRegs;
	wStatusBits : WORD;
	
	diEnergy : DINT;
	wEnergyArray : ARRAY [0..1] OF WORD;
	
	fbReadPower	: FB_MBReadRegs;
	diPower : DINT;
	wPowerArray : ARRAY [0..1] OF WORD;
	
	fbValues	: FB_MBReadRegs;
	
	fbReadOperationTime	: FB_MBReadRegs;
	diOperationTime : DINT;
	wOperationTimeArray : ARRAY [0..1] OF WORD;
	
	
	wValueArray : ARRAY [0..8] OF WORD;
END_VAR

//General
	offset := 0;
//Sekvens	
	bSekvensFlagga := oaksGVL.aBModbusSekvens[iModbusLoop] = UINT_TO_INT(nUnitID);
//Modbus konfiguering
	sIP := CONCAT (SIPAddr, '');
	sPort := CONCAT ('<br>Port: ', UINT_TO_STRING(nTCPPort)); 								
	sModbusID := CONCAT('<br>ID: ', UINT_TO_STRING(nUnitID));
	sModbusLoop := CONCAT('<br>Loop: ', INT_TO_STRING(iModbusLoop));	

	sTemp := sIP;
	sTemp := CONCAT(sTemp, sPort);
	sTemp := CONCAT(sTemp, sModbusID);
	sTemp := CONCAT(sTemp, sModbusLoop);
	
	PV8 := sTemp;

	fbStatusBits(
	sIPAddr:= sIpAddr, 
	nTCPPort:= nTCPPort, 
	nUnitID:= nUnitID, 
	nQuantity:= 1, 
	nMBAddr:= 200, 
	cbLength:= SIZEOF(wStatusBits), 
	pDestAddr:= ADR(wStatusBits), 
	bExecute:= bSekvensFlagga, 
	tTimeout:= T#1S, 
	bBusy=> , 
	bError=> , 
	nErrId=> , 
	cbRead=> );
	
	V := wStatusBits.6;
	AL := wStatusBits.10;
	AL1 := wStatusBits.11;
	AL2 := wStatusBits.12;
	
	fbReadPower(
	sIPAddr:= sIpAddr, 
	nTCPPort:= nTCPPort, 
	nUnitID:= nUnitID, 
	nQuantity:= 2, 
	nMBAddr:= 311, 
	cbLength:=SIZEOF(wPowerArray), 
	pDestAddr:= ADR(wPowerArray) , 
	bExecute:= bSekvensFlagga, 
	tTimeout:= T#1S, 
	bBusy=> , 
	bError=> , 
	nErrId=> , 
	cbRead=> );
	(* kWh to MWh *)
	diPower := ((wPowerArray[0] * 65535) + wPowerArray[1]);
	PV1 := DINT_TO_REAL(diPower);
	
	
	
	fbReadEnergy(
	sIPAddr:= sIpAddr, 
	nTCPPort:= nTCPPort, 
	nUnitID:= nUnitID, 
	nQuantity:= 2, 
	nMBAddr:= 331, 
	cbLength:=SIZEOF(wEnergyArray), 
	pDestAddr:= ADR(wEnergyArray) , 
	bExecute:= bSekvensFlagga, 
	tTimeout:= T#1S, 
	bBusy=> , 
	bError=> , 
	nErrId=> , 
	cbRead=> );
	(* kWh to MWh *)
	diEnergy := ((wEnergyArray[0] * 65535) + wEnergyArray[1]);
	PV := DINT_TO_REAL(diEnergy) / 1000;

	
	fbValues(
	sIPAddr:= sIpAddr, 
	nTCPPort:= nTCPPort, 
	nUnitID:= nUnitID, 
	nQuantity:= 9, 
	nMBAddr:= 300, 
	cbLength:=SIZEOF(wValueArray), 
	pDestAddr:= ADR(wValueArray) , 
	bExecute:= bSekvensFlagga, 
	tTimeout:= , 
	bBusy=> , 
	bError=> , 
	nErrId=> , 
	cbRead=> );
	
	rTemp := WORD_TO_REAL(wValueArray[0]);
	PV2 := rTemp / 10.0;
	rTemp := WORD_TO_REAL(wValueArray[1]);
	PV3 := rTemp / 10.0;
	PV4 := WORD_TO_REAL(wValueArray[3]);
	PV5 := WORD_TO_REAL(wValueArray[4]) *0.1;
	PV6:= WORD_TO_REAL(wValueArray[8]) *0.1;
	
(*	-1 
00327
00328
OperationTimeHI
OperationTimeLO Total operating time of the system. 1 hour
*)
	fbReadOperationTime(
	sIPAddr:= sIpAddr, 
	nTCPPort:= nTCPPort, 
	nUnitID:= nUnitID, 
	nQuantity:= 2, 
	nMBAddr:= 326, 
	cbLength:=SIZEOF(wOperationTimeArray), 
	pDestAddr:= ADR(wOperationTimeArray) , 
	bExecute:= bSekvensFlagga, 
	tTimeout:= T#1S, 
	bBusy=> , 
	bError=> , 
	nErrId=> , 
	cbRead=> );
	(* kWh to MWh *)
	diOperationTime := ((wOperationTimeArray[0] * 65535) + wOperationTimeArray[1]);
	PV7 := DINT_TO_REAL(diOperationTime);		
	
//Communication error
	fbKommTof(IN:=fbStatusBits.bError , PT:=T#20S , Q=> , ET=> );
	fbKommTon(bInput:=fbKommTof.Q , tAlarmDelay:=T#20M , bAutoReset:= , bAlarmOutput=> );
	FAULT :=fbKommTon.bAlarmOutput;
		
//Write busy	
	oaksgvl.aBModbusBusyFlagga[iModbusLoop,nUnitID] := fbStatusBits.bBusy OR fbReadPower.bBusy OR fbReadEnergy.bBusy OR fbValues.bBusy OR fbReadOperationTime.bBusy;

END_FUNCTION_BLOCK

// oaksModbusLibrary/Gruner/Givare/fbGrunerGTVMDD3MB
//OAKS AB
//2020-05-12
//Funktionsblock för läsning flöde via Gruner GT-VM-DD3-MB flödesmätare
FUNCTION_BLOCK fbGrunerGTVMDD3MB
VAR_INPUT
	sIPAddr : STRING := ''; 
	nTCPPort : UINT;
	nUnitID : UINT :=1;
	iModbusLoop : INT :=1; //Modbusslinga
			
END_VAR
VAR_OUTPUT
	
	PV AT %M* : REAL;//Flöde~wp:[unit]l/s[format]0[trendoptions]i:300
	FAULT AT %M* : BOOL;//Kommunikationsfel~wp:
	PV10 AT %M* : STRING;//Modbus konfigurering~wp:
	
END_VAR
VAR
	offset : WORD;
	rTemp : REAL;
	iTemp : UINT;
	bSekvensFlagga : BOOL;
	wAbsVolume : WORD;
		
	FB_MBReadRegs_ArrHolding1: FB_MBReadRegs;
	ArrHolding1 : ARRAY [0..10] OF WORD; //Holding
		
	//Kommunikationsfel
	fbKommTof : tof; 
	fbKommTon : ton;
	
	sIP: STRING(255);
	sPort: STRING(255);
	sModbusID: STRING(255);
	sModbusLoop: STRING(255);
	
	
	sTemp: STRING(255);
END_VAR

//General
	offset := 0;
//Sekvens	
	bSekvensFlagga := oaksGVL.aBModbusSekvens[iModbusLoop] = UINT_TO_INT(nUnitID);
//Modbus konfiguering
	sIP := CONCAT (SIPAddr, '');
	sPort := CONCAT ('<br>Port: ', UINT_TO_STRING(nTCPPort)); 								
	sModbusID := CONCAT('<br>ID: ', UINT_TO_STRING(nUnitID));
	sModbusLoop := CONCAT('<br>Loop: ', INT_TO_STRING(iModbusLoop));

	sTemp := sIP;
	sTemp := CONCAT(sTemp, sPort);
	sTemp := CONCAT(sTemp, sModbusID);
	sTemp := CONCAT(sTemp, sModbusLoop);
		
	PV10 := sTemp;
	
///////////////		
//READ
///////////////		
	
	//Read Holding 0-8
	FB_MBReadRegs_ArrHolding1(
	sIPAddr:= sIpAddr, 
	nTCPPort:= INT_TO_UINT(nTCPPort), 
	nUnitID:= INT_TO_BYTE(nUnitID), 
	nQuantity:= 8, 
	nMBAddr:= 0 + offset, 
	cbLength:= SIZEOF(ArrHolding1), 
	pDestAddr:= ADR(ArrHolding1), 
	bExecute:= bSekvensFlagga, 
	tTimeout:= T#3S, 
	bBusy=> , 
	bError=> , 
	nErrId=> , 
	cbRead=> );
	
		//Values
		//ArrHolding1[0]; //0
		//ArrHolding1[1]; //1
		//ArrHolding1[2]; //2
		//ArrHolding1[3]; //3
		//ArrHolding1[4]; //4
		//ArrHolding1[5]; //5
		//ArrHolding1[6]; //6
		wAbsVolume := ArrHolding1[7]; //7
							
		//Absolute Volume flow
		//Converter from m2 to l/s
		iTemp := WORD_TO_UINT(wAbsVolume);
		rTemp := UINT_TO_REAL(iTemp);
		PV := rTemp;
		
	
//Communication error
	fbKommTof(IN:=FB_MBReadRegs_ArrHolding1.bError , PT:=T#20S , Q=> , ET=> );
	fbKommTon(IN:=fbKommTof.Q , PT:=T#20M , Q=> , ET=> );
	FAULT :=fbKommTon.Q;
		
//Write busy	
	oaksgvl.aBModbusBusyFlagga[iModbusLoop,nUnitID] := FB_MBReadRegs_Arrholding1.bBusy;

END_FUNCTION_BLOCK

// oaksModbusLibrary/Gruner/Spjällställdon/fbGruner227CMXXMB
//OAKS AB
//2020-05-12
//Funktionsblock för styrning av spjällställdon utan flöde-/tryckmätning
FUNCTION_BLOCK fbGruner227CMXXMB
VAR_INPUT
	sIPAddr : STRING := ''; 
	nTCPPort : UINT;
	nUnitID : UINT :=1;
	iModbusLoop : INT :=1; //Modbusslinga
	rSetpoint : REAL;//Regulatorsignal	
		
END_VAR
VAR_OUTPUT
		
	OP AT %M* : REAL;//Relativ position~wp:[unit]%[format]0[trendoptions]i:300
	PV8 AT %M* : REAL;//Ställdonstyp:[format]0
	FAULT AT %M* : BOOL;//Kommunikationsfel~wp:
	PV10 AT %M* : STRING;//Modbus konfiguering~wp:
	
END_VAR
VAR
	offset : WORD;
	rTemp : REAL;
	iTemp : UINT;
	bSekvensFlagga : BOOL;
			
	FB_MBReadRegs_ArrHolding1: FB_MBReadRegs;
	ArrHolding1 : ARRAY [0..10] OF WORD; //Holding
	fbReadWriteHoldingReg_1: fbReadWriteHoldingReg;	
	
	//Kommunikationsfel
	fbKommTof : tof; 
	fbKommTon : ton;
	
	sIP: STRING(255);
	sPort: STRING(255);
	sModbusID: STRING(255);
	sModbusLoop: STRING(255);
	
	
	sTemp: STRING(255);
END_VAR

//General
	offset := 0;
//Sekvens	
	bSekvensFlagga := oaksGVL.aBModbusSekvens[iModbusLoop] = UINT_TO_INT(nUnitID);
//Modbus konfiguering
	sIP := CONCAT (SIPAddr, '');
	sPort := CONCAT ('<br>Port: ', UINT_TO_STRING(nTCPPort)); 								
	sModbusID := CONCAT('<br>ID: ', UINT_TO_STRING(nUnitID));
	sModbusLoop := CONCAT('<br>Loop: ', INT_TO_STRING(iModbusLoop));

	sTemp := sIP;
	sTemp := CONCAT(sTemp, sPort);
	sTemp := CONCAT(sTemp, sModbusID);
	sTemp := CONCAT(sTemp, sModbusLoop);
	
	PV10 := sTemp;
	
///////////////		
//READ
///////////////	
	
	//Read Holding 0-10
	FB_MBReadRegs_ArrHolding1(
	sIPAddr:= sIpAddr, 
	nTCPPort:= INT_TO_UINT(nTCPPort), 
	nUnitID:= INT_TO_BYTE(nUnitID), 
	nQuantity:= 6, 
	nMBAddr:= 0 + offset, 
	cbLength:= SIZEOF(ArrHolding1), 
	pDestAddr:= ADR(ArrHolding1), 
	bExecute:= bSekvensFlagga, 
	tTimeout:= T#3S, 
	bBusy=> , 
	bError=> , 
	nErrId=> , 
	cbRead=> );
	
		//Values
		//ArrHolding1[0]; //0 Setpoint 0.100%
		//ArrHolding1[1]; //1 Override command
		//ArrHolding1[2]; //2 Command
		
		iTemp := WORD_TO_UINT(ArrHolding1[3]); //3 Ställdons typ
		PV8 := UINT_TO_REAL(iTemp);
				
		//Relative Position
		iTemp := WORD_TO_UINT(ArrHolding1[4]); //4 Relativ position
		rTemp := UINT_TO_REAL(iTemp);
		OP := rTemp / 100;
				
		//ArrHolding1[5]; //5 Absolut position
		//ArrHolding1[6]; //6
		//ArrHolding1[7]; //7
		//ArrHolding1[8]; //8
		//ArrHolding1[8]; //9
		//ArrHolding1[8]; //10

///////////////		
//WRITE
///////////////			

rtemp := rSetpoint * 100;
iTemp := LIMIT(0,REAL_TO_UINT(rtemp ),10000);
		
//Write setpoint
fbReadWriteHoldingReg_1(
	sIPAddr:= sIpAddr, 
	nTCPPort:= INT_TO_UINT(nTCPPort), 
	nUnitID:= INT_TO_BYTE(nUnitID), 
	mBusAdr:= 0 + offset, 
	bEnable:= bSekvensFlagga, 
	iWrite:= iTemp, 
	iRead=> , 
	bError=> );
	
//Communication error
	fbKommTof(IN:=FB_MBReadRegs_ArrHolding1.bError , PT:=T#20S , Q=> , ET=> );
	fbKommTon(IN:=fbKommTof.Q , PT:=T#20M , Q=> , ET=> );
	FAULT :=fbKommTon.Q;
		
//Write busy	
	oaksgvl.aBModbusBusyFlagga[iModbusLoop,nUnitID] := FB_MBReadRegs_Arrholding1.bBusy OR fbReadWriteHoldingReg_1.bBusy;

END_FUNCTION_BLOCK

// oaksModbusLibrary/IMI hydronic/fbImiBrainCubeConnect
//OAKS AB
//2021-10-14
//Modbus block för IMI Hydronics BrainConnect expansionskärl
FUNCTION_BLOCK fbImiBrainCubeConnect
VAR_INPUT
	sIPAddr : STRING := ''; 
	nTCPPort : UINT;
	nUnitID : UINT :=1;
	iModbusLoop : INT :=1; //Modbusslinga
	tTimeout : TIME := T#20S;		
END_VAR
VAR_OUTPUT
	
	PV AT %M* : REAL;//Aktuellt tryck~wp:[unit]bar[format]0.0[trendoptions]i:300	
	PV1 AT %M* : REAL;//Aktuell nivå~wp:[unit]%[format]0[trendoptions]i:300	
	PV8 AT %M* : STRING;//Modbus konfiguering~wp:
	FAULT AT %M* : BOOL;//Kommunikationsfel~wp:
	
END_VAR
VAR
	offset : WORD;
	rTemp : REAL;
	iTemp : UINT;
	bSekvensFlagga : BOOL;
			
	FB_MBReadRegs_ArrHolding1: FB_MBReadRegs;
	ArrHolding1 : ARRAY [4..10] OF WORD; //Holding
		
	//Kommunikationsfel
	fbKommTof : tof; 
	fbKommTon : fbAlarm;
	
	sIP: STRING(255);
	sPort: STRING(255);
	sModbusID: STRING(255);
	sModbusLoop: STRING(255);
	sTemp : STRING(255);
	
	
END_VAR

//General
	offset := 0;
//Sekvens	
	bSekvensFlagga := oaksGVL.aBModbusSekvens[iModbusLoop] = UINT_TO_INT(nUnitID);
//Modbus konfiguering
	sIP := CONCAT (SIPAddr, '');
	sPort := CONCAT ('<br>Port: ', UINT_TO_STRING(nTCPPort)); 								
	sModbusID := CONCAT('<br>ID: ', UINT_TO_STRING(nUnitID));
	sModbusLoop := CONCAT('<br>Loop: ', INT_TO_STRING(iModbusLoop));	

	sTemp := sIP;
	sTemp := CONCAT(sTemp, sPort);
	sTemp := CONCAT(sTemp, sModbusID);
	sTemp := CONCAT(sTemp, sModbusLoop);
	
	PV8 := sTemp;

///////////////		
//READ
///////////////		
	
	//Read Holding 0-10
	FB_MBReadRegs_ArrHolding1(
	sIPAddr:= sIpAddr, 
	nTCPPort:= INT_TO_UINT(nTCPPort), 
	nUnitID:= INT_TO_BYTE(nUnitID), 
	nQuantity:= 2, 
	nMBAddr:= 516 + offset, 
	cbLength:= SIZEOF(ArrHolding1), 
	pDestAddr:= ADR(ArrHolding1), 
	bExecute:= bSekvensFlagga, 
	tTimeout:= tTimeout, 
	bBusy=> , 
	bError=> , 
	nErrId=> , 
	cbRead=> );
	
		//Values
		PV := fSignedConverter(rInput:= WORD_TO_REAL(ArrHolding1[4])) * 0.01; //4 Tryck (faktor 0.1)
		PV1 := fSignedConverter(rInput:= WORD_TO_REAL(ArrHolding1[5])) * 0.1; //5 Aktuell volym (faktor 1)
	
//Communication error
	fbKommTof(IN:=FB_MBReadRegs_ArrHolding1.bError , PT:=T#20S , Q=> , ET=> );
	fbKommTon(bInput:=fbKommTof.Q , tAlarmDelay:=T#20M , bAutoReset:= , bAlarmOutput=> );
	FAULT :=fbKommTon.bAlarmOutput;
		
//Write busy	
	oaksgvl.aBModbusBusyFlagga[iModbusLoop,nUnitID] := FB_MBReadRegs_Arrholding1.bBusy;

END_FUNCTION_BLOCK

// oaksModbusLibrary/Iv produkt/fbIvClimatixEnvistarIndication
FUNCTION_BLOCK fbIvClimatixEnvistarIndication
VAR_INPUT
	sIPAddr : STRING := ''; 
	nTCPPort : UINT := 502;
	nUnitID : UINT :=1;
	tTimeOut : TIME := T#20M;	
	tToggleTime : TIME := T#1s;
END_VAR
VAR_OUTPUT
		
	PV8 AT %M* : STRING;//Modbus konfiguering~wp:
	FAULT AT %M* : BOOL;//Kommunikationsfel~wp:
	
	HEAT_CIRCPUMP_V AT %M* : BOOL;//Driftindikering pump värme~wp:[trendoptions]i:14400, t:1
	COOL_CIRCPUMP_V AT %M* : BOOL;//Driftindikering pump kyla~wp:[trendoptions]i:14400, t:1
	
	SUPPLY_FAN_V AT %M* : BOOL;//Driftindikering tilluftsfläkt~wp:[trendoptions]i:14400, t:1
	SUPPLY_FAN_OP AT %M* : REAL;//Utsignal tilluftsfläkt~wp:[trendoptions]i:300	[unit]%[format]0
	EXHAUST_FAN_V AT %M* : BOOL;//Driftindikering frånluftsfläkt~wp:[trendoptions]i:14400, t:1
	EXHAUST_FAN_OP AT %M* : REAL;//Utsignal tilluftsfläkt~wp:[trendoptions]i:300[unit]%[format]0
END_VAR
VAR
	wHeatpump : WORD;
	wCoolpump : WORD;	

	rTemp : REAL;
	wSupfan : WORD;
	wExhfan : WORD;	

	fbToggle01 :	fbToggle;

	FB_MBReadInputRegsHeatpump : FB_MBReadInputRegs;
	FB_MBReadInputRegsCoolpump : FB_MBReadInputRegs;
	
	
	offset : WORD;
	iTemp : UINT;

		
	//Kommunikationsfel
	fbKommTof : tof; 
	fbKommTon : fbAlarm;
	
	sIP: STRING(255);
	sPort: STRING(255);
	sModbusID: STRING(255);
	sModbusLoop: STRING(255);
	sTemp : STRING(255);
	
	
	FB_MBReadInputRegsSupplyFan: FB_MBReadInputRegs;
	FB_MBReadInputRegsExhFan: FB_MBReadInputRegs;
END_VAR

//General
	offset := 0;
//Modbus konfiguering
	sIP := CONCAT (SIPAddr, '');
	sPort := CONCAT ('<br>Port: ', UINT_TO_STRING(nTCPPort)); 								
	sModbusID := CONCAT('<br>ID: ', UINT_TO_STRING(nUnitID));

	sTemp := sIP;
	sTemp := CONCAT(sTemp, sPort);
	sTemp := CONCAT(sTemp, sModbusID);
	
	PV8 := sTemp;
	fbToggle01(bStart:=TRUE , tTimeOn:=tToggleTime , tTimeOff:=tToggleTime , bOutput=> );

(*P11_V;;30041;INT;0;0;0;0;;0;Pump värme indikering;;i:300*)
	FB_MBReadInputRegsHeatpump(
	sIPAddr:= sIpAddr, 
	nTCPPort:= INT_TO_UINT(nTCPPort), 
	nUnitID:= INT_TO_BYTE(nUnitID), 
	nQuantity:= 1, 
	nMBAddr:= 40, 
	cbLength:=SIZEOF(wHeatpump) , 
	pDestAddr:=ADR(wHeatpump) , 
	bExecute:= fbToggle01.bOutput, 
	tTimeout:= T#3S, 
	bBusy=> , 
	bError=> , 
	nErrId=> , 
	cbRead=> );
	HEAT_CIRCPUMP_V := wHeatpump > 0;
//CP2_V;;30034;INT;0;0;0;0;;0;Pump kyla indikering;;i:300
	FB_MBReadInputRegsCoolpump(
	sIPAddr:= sIpAddr, 
	nTCPPort:= INT_TO_UINT(nTCPPort), 
	nUnitID:= INT_TO_BYTE(nUnitID), 
	nQuantity:= 1, 
	nMBAddr:= 33, 
	cbLength:=SIZEOF(wCoolpump) , 
	pDestAddr:=ADR(wCoolpump) , 
	bExecute:= fbToggle01.bOutput, 
	tTimeout:= T#3S, 
	bBusy=> , 
	bError=> , 
	nErrId=> , 
	cbRead=> );
	COOL_CIRCPUMP_V := wCoolpump > 0;
//TF_OP;;30029;INT;0;0;0;0;%;0;Tilluftsfläkt utsignal;;i:300
	FB_MBReadInputRegsSupplyFan(
	sIPAddr:= sIpAddr, 
	nTCPPort:= INT_TO_UINT(nTCPPort), 
	nUnitID:= INT_TO_BYTE(nUnitID), 
	nQuantity:=1 , 
	nMBAddr:= 28, 
	cbLength:=SIZEOF(wSupfan), 
	pDestAddr:=ADR(wSupfan) ,
	bExecute:= fbToggle01.bOutput, 
	tTimeout:= T#3S, 
	bBusy=> , 
	bError=> , 
	nErrId=> , 
	cbRead=> );
	
	rTemp := 	WORD_TO_REAL(wSupfan);
	SUPPLY_FAN_OP := rTemp;
	SUPPLY_FAN_V := wSupfan > 0;
//FF_OP;;30031;INT;0;0;0;0;%;0;Frånluftsfläkt utsignal;;i:300
	FB_MBReadInputRegsExhFan(
	sIPAddr:= sIpAddr, 
	nTCPPort:= INT_TO_UINT(nTCPPort), 
	nUnitID:= INT_TO_BYTE(nUnitID), 
	nQuantity:=1 , 
	nMBAddr:= 30, 
	cbLength:=SIZEOF(wExhfan), 
	pDestAddr:=ADR(wExhfan) ,
	bExecute:= fbToggle01.bOutput, 
	tTimeout:= T#3S, 
	bBusy=> , 
	bError=> , 
	nErrId=> , 
	cbRead=> );
	
	rTemp := 	WORD_TO_REAL(wExhfan);
	EXHAUST_FAN_OP := rTemp;
	EXHAUST_FAN_V := wSupfan > 0;

//Communication error
	fbKommTof(IN:=FB_MBReadInputRegsHeatpump.bError , PT:=T#20S , Q=> , ET=> );
	fbKommTon(bInput:=fbKommTof.Q , tAlarmDelay:=tTimeOut , bAutoReset:= , bAlarmOutput=> );
	FAULT :=fbKommTon.bAlarmOutput;

END_FUNCTION_BLOCK

// oaksModbusLibrary/Iv produkt/fbIvClimatixEnvistarOperationLevel
FUNCTION_BLOCK fbIvClimatixEnvistarOperationLevel
VAR_INPUT
	sIPAddr : STRING; // Ip-adress till iv-aggregat
	usiTimechannel : USINT := 3; // Välj hastighet vid tidkanal 0-4 Auto*Off*Stage 1*Stage 2*Stage 3
	bTimechannel : BOOL; // Ingång för knytning av tidkanal
	usiPushbutton : USINT := 3; // Välj hastighet vid tryckknappsdrift 0-4 Auto*Off*Stage 1*Stage 2*Stage 3
	bPushbutton : BOOL; // Ingång för knytning av tryckkanpp för förlängd drift
	usiPrescence : USINT := 2; // Välj hastighet vid närvarodrift 0-4 Auto*Off*Stage 1*Stage 2*Stage 3
	bPrescence : BOOL; // Ingång för knytning av närvarosensor eller valfritt. Bara att lämna den tom om den ej används.
END_VAR
VAR_OUTPUT
	PV8 : STRING; //Modbus konfiguering~wp:
	FAULT AT %M* : BOOL;//Kommunikationsfel Iv produkt Climatix Ventilationsaggregat~wp:
END_VAR
VAR
	//Kommunikationsfel
	fbKommTof : tof; 
	fbAlarmCommunicationError : fbAlarm;
	fbToggle_run: fbToggle;
	fbReadWriteHoldingIvProduktClimatixEnvistarHoldingRegAdr792 : fbReadWriteHoldingReg;
END_VAR
VAR PERSISTENT
	tToggleTid : TIME := T#3S;
END_VAR
VAR // added by the converter: edge detectors and wires of the graphical bodies
    _w1, _w3 : ANY;
    _w2 : BOOL;
END_VAR

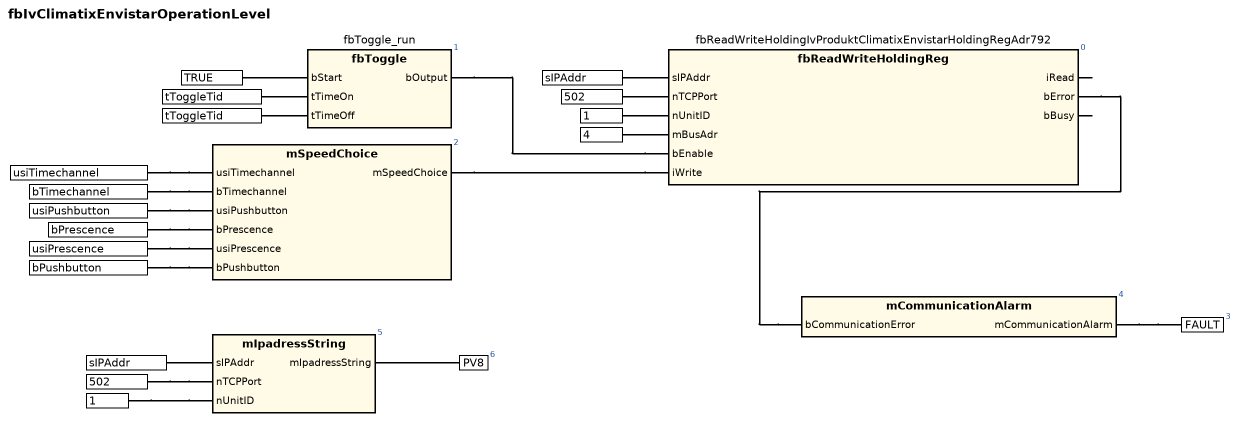
// note: 6 stored wires end on pins the file does not list and are not shown
fbReadWriteHoldingIvProduktClimatixEnvistarHoldingRegAdr792(
    sIPAddr := sIPAddr,
    nTCPPort := 502,
    nUnitID := 1,
    mBusAdr := 4,
    bEnable := fbToggle_run.bOutput,
    iWrite := _w1); // fbReadWriteHoldingReg
fbToggle_run(bStart := TRUE, tTimeOn := tToggleTid, tTimeOff := tToggleTid); // fbToggle
_w1 := mSpeedChoice(usiTimechannel := usiTimechannel, bTimechannel := bTimechannel, usiPushbutton := usiPushbutton, bPrescence := bPrescence, usiPrescence := usiPrescence, bPushbutton := bPushbutton);
FAULT := _w2;
_w2 := mCommunicationAlarm(bCommunicationError := fbReadWriteHoldingIvProduktClimatixEnvistarHoldingRegAdr792.bError);
_w3 := mIpadressString(sIPAddr := sIPAddr, nTCPPort := 502, nUnitID := 1);
PV8 := _w3;

METHOD mCommunicationAlarm : BOOL
VAR_INPUT
	bCommunicationError : BOOL;
END_VAR
VAR 

	
END_VAR
	//Communication error
	fbKommTof(IN:=bCommunicationError , PT:=T#20S , Q=> , ET=> );
	fbAlarmCommunicationError(bInput:=fbKommTof.Q , tAlarmDelay:=T#60S , bAutoReset:=TRUE , bAlarmOutput=> );
	mCommunicationAlarm :=fbAlarmCommunicationError.bAlarmOutput;
END_METHOD

METHOD mIpadressString : STRING
VAR_INPUT
	sIPAddr : STRING := ''; 
	nTCPPort : UINT;
	nUnitID : UINT :=1;
END_VAR
VAR
	sIP: STRING(255);
	sPort: STRING(255);
	sModbusID: STRING(255);
	sTemp : STRING(255);
END_VAR
//Modbus konfiguering
	sIP := CONCAT (SIPAddr, '');
	sPort := CONCAT ('<br>Port: ', UINT_TO_STRING(nTCPPort)); 								
	sModbusID := CONCAT('<br>ID: ', UINT_TO_STRING(nUnitID));

	sTemp := sIP;
	sTemp := CONCAT(sTemp, sPort);
	sTemp := CONCAT(sTemp, sModbusID);
	
	mIpadressString := sTemp;
END_METHOD

METHOD PRIVATE mSpeedChoice : USINT
VAR_INPUT
	usiTimechannel : USINT;
	bTimechannel : BOOL;
	usiPushbutton : USINT;
	bPushbutton : BOOL;
	usiPrescence : USINT;
	bPrescence : BOOL;
END_VAR
IF bTimechannel THEN
	mSpeedChoice := usiTimechannel;
ELSIF bPushbutton THEN
	mSpeedChoice := usiPushbutton;	
ELSIF bPrescence THEN
	mSpeedChoice := usiPrescence;	
ELSE 
	mSpeedChoice := 1;
END_IF
END_METHOD

END_FUNCTION_BLOCK

// oaksModbusLibrary/Iv produkt/fbIvSaphirOperationLevel
FUNCTION_BLOCK fbIvSaphirOperationLevel
VAR_INPUT
	sIPAddr : STRING; // Ip-adress till iv-aggregat
	nTCPPort : UINT := 502;
	nUnitID : UINT :=1;
	usiTimechannel : USINT := 4; // Välj hastighet vid tidkanal 0 = Internal time , 1= Off, 2 = Eco St1 3 = Eco St2, 4 = Comf St1, 5 = Comf St2
	bTimechannel : BOOL; // Ingång för knytning av tidkanal
	usiPushbutton : USINT := 4; // Välj hastighet vid tryckknappsdrift 0 = Internal time , 1= Off, 2 = Eco St1 3 = Eco St2, 4 = Comf St1, 5 = Comf St2
	bPushbutton : BOOL; // Ingång för knytning av tryckkanpp för förlängd drift
	usiPrescence : USINT := 4; // Välj hastighet vid närvarodrift 0 = Internal time , 1= Off, 2 = Eco St1 3 = Eco St2, 4 = Comf St1, 5 = Comf St2
	bPrescence : BOOL; // Ingång för knytning av närvarosensor eller valfritt. Bara att lämna den tom om den ej används.
END_VAR
VAR_OUTPUT
	PV8 : STRING := ''; //Modbus konfiguering~wp:
	FAULT AT %M* : BOOL;//Kommunikationsfel Iv produkt Saphir Ventilationsaggregat~wp:
END_VAR
VAR
	//Kommunikationsfel
	fbKommTof : tof; 
	fbAlarmCommunicationError : fbAlarm;
	fbToggle_run: fbToggle;
	fbReadWriteHoldingIvProduktSaphir : fbReadWriteHoldingReg;
END_VAR
VAR PERSISTENT
	tToggleTid : TIME := T#3S;
END_VAR
VAR // added by the converter: edge detectors and wires of the graphical bodies
    _w1, _w3 : ANY;
    _w2 : BOOL;
END_VAR

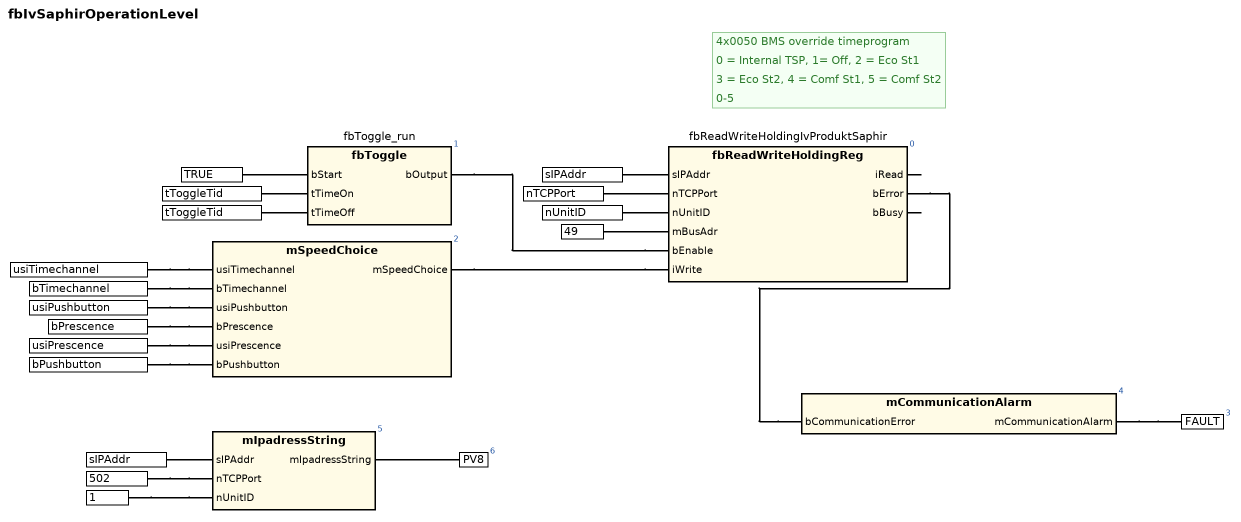
// note: 6 stored wires end on pins the file does not list and are not shown
// 4x0050 BMS override timeprogram
// 0 = Internal TSP, 1= Off, 2 = Eco St1
// 3 = Eco St2, 4 = Comf St1, 5 = Comf St2
// 0-5
fbReadWriteHoldingIvProduktSaphir(
    sIPAddr := sIPAddr,
    nTCPPort := nTCPPort,
    nUnitID := nUnitID,
    mBusAdr := 49,
    bEnable := fbToggle_run.bOutput,
    iWrite := _w1); // fbReadWriteHoldingReg
fbToggle_run(bStart := TRUE, tTimeOn := tToggleTid, tTimeOff := tToggleTid); // fbToggle
_w1 := mSpeedChoice(usiTimechannel := usiTimechannel, bTimechannel := bTimechannel, usiPushbutton := usiPushbutton, bPrescence := bPrescence, usiPrescence := usiPrescence, bPushbutton := bPushbutton);
FAULT := _w2;
_w2 := mCommunicationAlarm(bCommunicationError := fbReadWriteHoldingIvProduktSaphir.bError);
_w3 := mIpadressString(sIPAddr := sIPAddr, nTCPPort := 502, nUnitID := 1);
PV8 := _w3;

METHOD mCommunicationAlarm : BOOL
VAR_INPUT
	bCommunicationError : BOOL;
END_VAR
VAR 

	
END_VAR
	//Communication error
	fbKommTof(IN:=bCommunicationError , PT:=T#20S , Q=> , ET=> );
	fbAlarmCommunicationError(bInput:=fbKommTof.Q , tAlarmDelay:=T#60S , bAutoReset:=TRUE , bAlarmOutput=> );
	mCommunicationAlarm :=fbAlarmCommunicationError.bAlarmOutput;
END_METHOD

METHOD mIpadressString : STRING
VAR_INPUT
	sIPAddr : STRING := ''; 
	nTCPPort : UINT;
	nUnitID : UINT :=1;
END_VAR
VAR
	sIP: STRING(255);
	sPort: STRING(255);
	sModbusID: STRING(255);
	sTemp : STRING(255);
END_VAR
//Modbus konfiguering
	sIP := CONCAT (SIPAddr, '');
	sPort := CONCAT ('<br>Port: ', UINT_TO_STRING(nTCPPort)); 								
	sModbusID := CONCAT('<br>ID: ', UINT_TO_STRING(nUnitID));

	sTemp := sIP;
	sTemp := CONCAT(sTemp, sPort);
	sTemp := CONCAT(sTemp, sModbusID);
	
	mIpadressString := sTemp;
END_METHOD

METHOD PRIVATE mSpeedChoice : USINT
VAR_INPUT
	usiTimechannel : USINT;
	bTimechannel : BOOL;
	usiPushbutton : USINT;
	bPushbutton : BOOL;
	usiPrescence : USINT;
	bPrescence : BOOL;
END_VAR
IF bTimechannel THEN
	mSpeedChoice := usiTimechannel;
ELSIF bPushbutton THEN
	mSpeedChoice := usiPushbutton;	
ELSIF bPrescence THEN
	mSpeedChoice := usiPrescence;	
ELSE 
	mSpeedChoice := 1;
END_IF
END_METHOD

END_FUNCTION_BLOCK

// oaksModbusLibrary/IVT/fbIvtRego5200BorVarde
//OAKS AB
//2020-05-12
//Börvärdesblock för att skriva till Ivt värmepump med Rego 5200 
FUNCTION_BLOCK fbIvtRego5200BorVarde EXTENDS fbSetPointOutdoorCompC
VAR_INPUT
	sIPAddr : STRING := ''; 
	nTCPPort : UINT;
	nUnitID : UINT :=1;
			
END_VAR
VAR_OUTPUT
	PV4 AT %M*: REAL; //Utetemperatur~wp:[unit]°C[format]0.0	

	PV AT %M*: REAL; //Framledningstemperatur~wp:[unit]°C[format]0.0
	PV8 AT %M* : STRING;//Modbus konfiguering~wp:
	AL8 AT %M* : BOOL;//Kommunikationsfel~wp:
	
END_VAR
VAR
	rPvTemp : REAL;
	rPv4Temp : REAL;
	bWatchDog : BOOL;	

	fbToggle01 : fbToggle;
	
	FB_MBReadInputRegsProcessValue,FB_MBReadInputRegsOutdoortemp : FB_MBReadInputRegs;
	ProcessValueWord : WORD;
	OutdoorTempWord : WORD;
	
	fbReadWriteHoldingRegSetpoint :fbReadWriteHoldingReg;

	offset : WORD;
	rTemp : REAL;
	iTemp : UINT;


	//Kommunikationsfel
	fbKommTof : tof; 
	fbKommTon : fbAlarm;
	
	sIP: STRING(255);
	sPort: STRING(255);
	sModbusID: STRING(255);
	sTemp : STRING(255);
	FB_MBWriteCoilsWatchdog,FB_MBWriteCoilsEnableExternalFlowSetpoint: FB_MBWriteCoils;
END_VAR

	SUPER^();
//General
	offset := 0;

//Modbus konfiguering
	sIP := CONCAT (SIPAddr, '');
	sPort := CONCAT ('<br>Port: ', UINT_TO_STRING(nTCPPort)); 								
	sModbusID := CONCAT('<br>ID: ', UINT_TO_STRING(nUnitID));

	sTemp := sIP;
	sTemp := CONCAT(sTemp, sPort);
	sTemp := CONCAT(sTemp, sModbusID);
	
	PV8 := sTemp;

	
	fbToggle01(bStart:=TRUE  , tTimeOn:=T#1S , tTimeOff:=T#1S , bOutput=> );
///////////////		
//READ
///////////////		

// T0 framledningsgivare : 30011
	FB_MBReadInputRegsProcessValue(
	sIPAddr:= sIpAddr, 
	nTCPPort:= INT_TO_UINT(nTCPPort), 
	nUnitID:= INT_TO_BYTE(nUnitID), 
	nQuantity:= 1, 
	nMBAddr:=10 , 
	cbLength:= SIZEOF(ProcessValueWord), 
	pDestAddr:=ADR(ProcessValueWord) , 
	bExecute:= fbToggle01.bOutput, 
	tTimeout:= , 
	bBusy=> , 
	bError=> , 
	nErrId=> , 
	cbRead=> );
	rPvTemp := fSignedConverter(WORD_TO_REAL(ProcessValueWord));
	PV := rPvTemp / 10;
	
	
	FB_MBReadInputRegsOutdoortemp(
	sIPAddr:= sIpAddr, 
	nTCPPort:= INT_TO_UINT(nTCPPort), 
	nUnitID:= INT_TO_BYTE(nUnitID), 
	nQuantity:= 1, 
	nMBAddr:=12 , 
	cbLength:= SIZEOF(OutdoorTempWord), 
	pDestAddr:=ADR(OutdoorTempWord) , 
	bExecute:= fbToggle01.bOutput, 
	tTimeout:= , 
	bBusy=> , 
	bError=> , 
	nErrId=> , 
	cbRead=> );
	rPv4Temp := fSignedConverter(WORD_TO_REAL(OutdoorTempWord));
	PV4 := rPv4Temp / 10;
///////////////		
//WRITE
///////////////	
// Skriv önskat börvärde till adress 40053
	iTemp := REAL_TO_UINT(CSP) * 10; 
	fbReadWriteHoldingRegSetpoint(
	sIPAddr:= sIpAddr, 
	nTCPPort:= INT_TO_UINT(nTCPPort), 
	nUnitID:= INT_TO_BYTE(nUnitID), 
	mBusAdr:= 52, 
	bEnable:=fbToggle01.bOutput , 
	iWrite:=iTemp , 
	iRead=> , 
	bError=> , 
	bBusy=> );
// Nollställ watchdog minst var 5e minut genom att sätta adress 5 till 1.
	bWatchDog := TRUE;
	FB_MBWriteCoilsWatchdog(
	sIPAddr:= sIpAddr, 
	nTCPPort:= INT_TO_UINT(nTCPPort), 
	nUnitID:= INT_TO_BYTE(nUnitID), 
	nQuantity:=1 , 
	nMBAddr:=4 , 
	cbLength:= SIZEOF(bWatchDog), 
	pSrcAddr:=ADR(bWatchDog) , 
	bExecute:=fbToggle01.bOutput , 
	tTimeout:= , 
	bBusy=> , 
	bError=> , 
	nErrId=> );
// Aktivera funktionen External flow setpoint genom att sätta adress 8 till 1	
	FB_MBWriteCoilsEnableExternalFlowSetpoint(
	sIPAddr:= sIpAddr, 
	nTCPPort:= INT_TO_UINT(nTCPPort), 
	nUnitID:= INT_TO_BYTE(nUnitID), 
	nQuantity:=1 , 
	nMBAddr:=7 , 
	cbLength:= SIZEOF(bWatchDog), 
	pSrcAddr:=ADR(bWatchDog) , 
	bExecute:=fbToggle01.bOutput , 
	tTimeout:= , 
	bBusy=> , 
	bError=> , 
	nErrId=> );
//Communication error
	fbKommTof(IN:=FB_MBReadInputRegsProcessValue.bError , PT:=T#20S , Q=> , ET=> );
	fbKommTon(bInput:=fbKommTof.Q , tAlarmDelay:=T#20M , bAutoReset:= , bAlarmOutput=> );
	AL8 :=fbKommTon.bAlarmOutput;

END_FUNCTION_BLOCK

// oaksModbusLibrary/Metz/Givare/fbMetzMR_AI8GeneralSensor
FUNCTION_BLOCK fbMetzMR_AI8GeneralSensor
//OAKS AB
//2022-06-01
//Generellt givarblock för Metz IO med givarfel och handställningsmöjlighet.
VAR_INPUT
sensor : ST_MetzAI8Sensor;
rSensorErrorMin : REAL := -50; //Min. begränsning givarfel
rSensorErrorMax : REAL := 50; //Max. begränsning givarfel
 
END_VAR
VAR_OUTPUT
	rOutput : REAL;//Utgång knyts till tagg
	{attribute 'OPC.UA.DA' := '1'}
	PV8 AT %M* : STRING := '';  //Givartyp~wp:[trendoptions]i:14400, t:1	
	{attribute 'OPC.UA.DA' := '1'}
	FAULT AT %M* : BOOL := FALSE;//Givarfel~wp:
	{attribute 'OPC.UA.DA' := '1'}
	AL8 AT %M* : BOOL := FALSE; //Givare handställd~wp:[alarmoptions]p:3
END_VAR
VAR
	bSensorErrorInternal : BOOL; //Sensorfel aktiverat 
	fbAlarm_SensorError: fbAlarm;
	tSensorErrorDelay : TIME := T#30S;
	rTemp: REAL;
END_VAR
VAR_INPUT PERSISTENT 
	{attribute 'OPC.UA.DA' := '1'}
	M AT %M* : BOOL;//Handställning~wp:
	rHandsetValue : REAL; //OPM värde
	rX1 : REAL := 0; //Råvärde 1
	rX2 : REAL := 10; //Råvärde 2
	rY1 : REAL := 0; //Mätvärde 1
	rY2 : REAL := 0; //Mätvärde 2	
END_VAR

//Scale
rTemp := fScale2p(sensor.rRawValue, rY1, rY2, rX1, rX2);

//Manual alarm
	AL8 := M;

//Manual output
	IF M THEN
		rOutput := rHandsetValue;
	ELSIF FAULT THEN
		rOutput := LIMIT(rSensorErrorMin, sensor.rRawValue,rSensorErrorMax);
	ELSE 
		rOutput := rTemp;
	END_IF
	
//Sensor fault
IF (sensor.rRawValue >= rSensorErrorMax) OR (sensor.rRawValue <= rSensorErrorMin) THEN
	bSensorErrorInternal := TRUE;
ELSE 
	bSensorErrorInternal := FALSE;
END_IF

fbAlarm_SensorError(bInput:= bSensorErrorInternal OR sensor.bComError, tAlarmDelay:= tSensorErrorDelay, bAutoReset:= TRUE, bAlarmOutput=> );

FAULT := sensor.bComError OR fbAlarm_SensorError.bAlarmOutput;

//Sensor info
PV8 := sensor.sSensorConfig;

END_FUNCTION_BLOCK

// oaksModbusLibrary/Metz/Givare/fbMetzMR_AI8TempSensor
FUNCTION_BLOCK fbMetzMR_AI8TempSensor
//OAKS AB
//2022-06-01
//Givarblock för temperaturgivare Metz IO med givarfel och handställningsmöjlighet.
VAR_INPUT
 sensor : ST_MetzAI8Sensor;
 rSensorErrorMin : REAL := -50; //Min. begränsning givarfel
 rSensorErrorMax : REAL := 50; //Max. begränsning givarfel
END_VAR
VAR_OUTPUT
	{attribute 'OPC.UA.DA' := '1'}
	PV AT %M* : REAL;//Temperatur~wp:[unit]°C[format]0.0[trendoptions]i:300
	{attribute 'OPC.UA.DA' := '1'}
	PV8 AT %M* : STRING := '';  //Givartyp~wp:[trendoptions]i:14400, t:1	
	{attribute 'OPC.UA.DA' := '1'}
	FAULT AT %M* : BOOL := FALSE;//Givarfel~wp:
	{attribute 'OPC.UA.DA' := '1'}
	AL8 AT %M* : BOOL := FALSE; //Givare handställd~wp:[alarmoptions]p:3
END_VAR
VAR
	bSensorErrorInternal : BOOL; //Sensorfel aktiverat 
	fbAlarm_SensorError: fbAlarm;
	tSensorErrorDelay : TIME := T#30S;
END_VAR
VAR_INPUT PERSISTENT 
	{attribute 'OPC.UA.DA' := '1'}
	M AT %M* : BOOL;//Handställning~wp:
	{attribute 'OPC.UA.DA' := '1'}
	OPM AT %M* : REAL;//Värde handställning~wp:[unit]°C[format]0.0
END_VAR

//Manual alarm
	AL8 := M;

//Manual output
	IF M THEN
		PV := OPM;
	ELSIF FAULT THEN
		PV := LIMIT(rSensorErrorMin, sensor.rRawValue,rSensorErrorMax);
	ELSE 
		PV := sensor.rRawValue;
	END_IF
	
//Sensor fault
IF (sensor.rRawValue >= rSensorErrorMax) OR (sensor.rRawValue <= rSensorErrorMin) THEN
	bSensorErrorInternal := TRUE;
ELSE 
	bSensorErrorInternal := FALSE;
END_IF

fbAlarm_SensorError(bInput:= bSensorErrorInternal OR sensor.bComError, tAlarmDelay:= tSensorErrorDelay, bAutoReset:= TRUE, bAlarmOutput=> );

FAULT := sensor.bComError OR fbAlarm_SensorError.bAlarmOutput;

//Sensor info
PV8 := sensor.sSensorConfig;

END_FUNCTION_BLOCK

// oaksModbusLibrary/Metz/fbMetzMR_AI8
//Oaks AB
//2022-05-13 / Johan Bornemyr
//Funktionsblock för hantering av Metz MR IO-system. 
//MR-AI8. Modul med 8 Analoga ingångar för resistans och 0-10V.
//Utgångsvärden knyts mot variabel med SI-enhet. 
FUNCTION_BLOCK fbMetzMR_AI8
VAR_INPUT
	bEnable : BOOL := TRUE; //Aktivering
	modbusTCP : ST_ModbusTCP;
	nUnitID: BYTE := 0;
END_VAR

VAR_INPUT PERSISTENT
	sensor1config : ST_MetzAI8config;
	sensor2config : ST_MetzAI8config;
	sensor3config : ST_MetzAI8config;
	sensor4config : ST_MetzAI8config;
	sensor5config : ST_MetzAI8config;
	sensor6config : ST_MetzAI8config;
	sensor7config : ST_MetzAI8config;
	sensor8config : ST_MetzAI8config;
END_VAR

VAR_OUTPUT
	AI1_PV AT %M* : REAL; //Råvärde utgång 1~wp:[format]0.00
	AI1_PV1 AT %M* : STRING;//Konfigurering ingång 1~wp:
	sensor1 : ST_MetzAI8Sensor; //Skicka till sensorblock
	AI2_PV AT %M* : REAL; //Råvärde utgång 2~wp:[format]0.00
	AI2_PV1 AT %M* : STRING;//Konfigurering ingång 2~wp:
	sensor2 : ST_MetzAI8Sensor; //Skicka till sensorblock
	AI3_PV AT %M* : REAL; //Råvärde utgång 3~wp:[format]0.00
	AI3_PV1 AT %M* : STRING;//Konfigurering ingång 3~wp:
	sensor3 : ST_MetzAI8Sensor; //Skicka till sensorblock
	AI4_PV AT %M* : REAL; //Råvärde utgång 4~wp:[format]0.00
	AI4_PV1 AT %M* : STRING;//Konfigurering ingång 4~wp:
	sensor4 : ST_MetzAI8Sensor; //Skicka till sensorblock
	AI5_PV AT %M* : REAL; //Råvärde utgång 5~wp:[format]0.00
	AI5_PV1 AT %M* : STRING;//Konfigurering ingång 5~wp:
	sensor5 : ST_MetzAI8Sensor; //Skicka till sensorblock
	AI6_PV AT %M* : REAL; //Råvärde utgång 6~wp:[format]0.00
	AI6_PV1 AT %M* : STRING;//Konfigurering ingång 6~wp:
	sensor6 : ST_MetzAI8Sensor; //Skicka till sensorblock
	AI7_PV AT %M* : REAL; //Råvärde utgång 7~wp:[format]0.00
	AI7_PV1 AT %M* : STRING;//Konfigurering ingång 7~wp:
	sensor7 : ST_MetzAI8Sensor; //Skicka till sensorblock
	AI8_PV AT %M* : REAL; //Råvärde utgång 8~wp:[format]0.00
	AI8_PV1 AT %M* : STRING;//Konfigurering ingång 8~wp:
	sensor8 : ST_MetzAI8Sensor; //Skicka till sensorblock
	
	PV8 AT %M* : STRING;//Modbus konfiguering~wp:
	FAULT AT %M* : BOOL;//Kommunikationsfel~wp:
	
END_VAR
VAR
	sIP: STRING(255);
	sPort: STRING(255);
	sModbusID: STRING(255);
	sModbusLoop: STRING(255);
	sTemp : STRING(255);
	tTimeOut : TIME :=T#5S;
	iStep: INT;
	bError: BOOL;
	bBusy: BOOL;	
	bSekvensFlagga : BOOL;
	

	
	//Configuration
	FB_MBReadInputRegs_Values: FB_MBReadInputRegs;
	wInputRegs1 : ARRAY[0..15] OF WORD; //Läs input regs modbus function 4.
	wInputRegs2w : ARRAY[16..23] OF WORD; //Läs/skriv input regs modbus function 16.
	wInputRegs2r : ARRAY[16..23] OF WORD; //Läs/skriv input regs modbus function 16.
	
	FB_MBWriteRegs_Config: FB_MBWriteRegs;
	FB_MBReadRegs_Config: FB_MBReadRegs;
	arrIndex: INT;
	iConfigChanged: INT;
	bChangeConfig: BOOL;
		
	//Communication error
	fbKommTof : tof; 
	fbKommTon : fbAlarm;

	//Convert to float
	rTempArr: ARRAY[0..1] OF WORD;
	rTemp: REAL;
	R_TRIG_Sekvens: R_TRIG;
	
END_VAR

//Sekvens	
	R_TRIG_Sekvens(CLK:= oaksGVL.aBModbusSekvens[modbusTCP.iModbusLoop] = BYTE_TO_INT(nUnitID), Q=> bSekvensFlagga);
	
//Modbus config
	sIP := CONCAT (modbusTCP.sIPAddr, '');
	sPort := CONCAT ('<br>Port: ', UINT_TO_STRING(modbusTCP.nTCPPort)); 								
	sModbusID := CONCAT('<br>ID: ', BYTE_TO_STRING(nUnitID));
	sModbusLoop := CONCAT('<br>Loop: ', INT_TO_STRING(modbusTCP.iModbusLoop));	

	sTemp := sIP;
	sTemp := CONCAT(sTemp, sPort);
	sTemp := CONCAT(sTemp, sModbusID);
	sTemp := CONCAT(sTemp, sModbusLoop);
	
	PV8 := sTemp;

	CASE iStep OF

	0: 	//Start/reset
		bBusy := FALSE;
				
		IF bEnable AND bSekvensFlagga THEN
			iStep := 1;
			bError := FALSE;
		END_IF
		
	1: 	//Read measured values
		bBusy := TRUE;
			
		FB_MBReadInputRegs_Values.bExecute := TRUE;
	
		FB_MBReadInputRegs_Values(
		sIPAddr:= modbusTCP.sIpAddr, 
		nTCPPort:= modbusTCP.nTCPPort, 
		nUnitID:= nUnitID, 
		nQuantity:= 16,
		nMBAddr:= 0, 
		cbLength:= SIZEOF(wInputRegs1), 
		pDestAddr:= ADR(wInputRegs1), 
		bExecute:= , 
		tTimeout:= tTimeOut, 
		bBusy=> , 
		bError=> , 
		nErrId=> , 
		cbRead=> );
		
		//Ingång 1
		rTempArr[0] := wInputRegs1[1];
		rTempArr[1] := wInputRegs1[0]; 
	 	rTemp := fWordToReal(rTempArr);
		
		AI1_PV := fWordToReal(rTempArr);
		
		IF sensor1config.bResistance THEN
			AI1_PV := fWordToReal(rTempArr);
			AI1_PV1 := CONCAT('Givartyp: ', TO_STRING(sensor1config.sensorType));
		ELSE
			stemp := '0-10V';
			AI1_PV1 := sTemp;
		END_IF
		
		//Info till sensorblock
		sensor1.bComError := FAULT;
		sensor1.rRawValue := AI1_PV;
		sensor1.sSensorConfig := AI1_PV1;
		
		//Ingång 2
		rTempArr[0] := wInputRegs1[3];
		rTempArr[1] := wInputRegs1[2];
		rTemp := fWordToReal(rTempArr);
		
		AI2_PV := fWordToReal(rTempArr);
		
		IF sensor2config.bResistance THEN
			AI2_PV1 := CONCAT('Givartyp: ', TO_STRING(sensor2config.sensorType));
		ELSE
			stemp := '0-10V';
			AI2_PV1 := sTemp; 
  
		END_IF
		
		//Info till sensorblock
		sensor2.bComError := FAULT;
		sensor2.rRawValue := AI2_PV;
		sensor2.sSensorConfig := AI2_PV1;
		
		//Ingång 3
		rTempArr[0] := wInputRegs1[5];
		rTempArr[1] := wInputRegs1[4];
		rTemp := fWordToReal(rTempArr);
		
		AI3_PV := fWordToReal(rTempArr);
		
		IF sensor3config.bResistance THEN
			AI3_PV1 := CONCAT('Givartyp: ', TO_STRING(sensor3config.sensorType));
		ELSE
			stemp := '0-10V';
			AI3_PV1 := sTemp; 
		END_IF
		
		//Info till sensorblock
		sensor3.bComError := FAULT;
		sensor3.rRawValue := AI3_PV;
		sensor3.sSensorConfig := AI3_PV1;
		
		//Ingång 4
		rTempArr[0] := wInputRegs1[7];
		rTempArr[1] := wInputRegs1[6];
		rTemp := fWordToReal(rTempArr);
		
		AI4_PV := fWordToReal(rTempArr);
		
		IF sensor4config.bResistance THEN
			AI4_PV1 := CONCAT('Givartyp: ', TO_STRING(sensor4config.sensorType));
		ELSE
			stemp := '0-10V';
			AI4_PV1 := sTemp;
		END_IF
		
		//Info till sensorblock
		sensor4.bComError := FAULT;
		sensor4.rRawValue := AI4_PV;
		sensor4.sSensorConfig := AI4_PV1;
		
		//Ingång 5
		rTempArr[0] := wInputRegs1[9];
		rTempArr[1] := wInputRegs1[8];
		rTemp := fWordToReal(rTempArr);

		AI5_PV := fWordToReal(rTempArr);
	
		IF sensor5config.bResistance THEN
			AI5_PV1 := CONCAT('Givartyp: ', TO_STRING(sensor5config.sensorType));
		ELSE
			stemp := '0-10V';
			AI5_PV1 := sTemp;
		END_IF
		
		//Info till sensorblock
		sensor5.bComError := FAULT;
		sensor5.rRawValue := AI5_PV;
		sensor5.sSensorConfig := AI5_PV1;
		
		//Ingång 6
		rTempArr[0] := wInputRegs1[11];
		rTempArr[1] := wInputRegs1[10]; 
		rTemp := fWordToReal(rTempArr);
		
		AI6_PV := fWordToReal(rTempArr);
				
		IF sensor6config.bResistance THEN
			AI6_PV1 := CONCAT('Givartyp: ', TO_STRING(sensor6config.sensorType));
		ELSE
			stemp := '0-10V';
			AI6_PV1 := sTemp;
		END_IF
		
		//Info till sensorblock
		sensor6.bComError := FAULT;
		sensor6.rRawValue := AI6_PV;
		sensor6.sSensorConfig := AI6_PV1;
		
		//Ingång 7
		rTempArr[0] := wInputRegs1[13];
		rTempArr[1] := wInputRegs1[12];
		rTemp := fWordToReal(rTempArr);
		
		AI7_PV := fWordToReal(rTempArr);
		
		IF sensor7config.bResistance THEN
			
			AI7_PV1 := CONCAT('Givartyp: ', TO_STRING(sensor7config.sensorType));
		ELSE
			stemp := '0-10V';
			AI7_PV1 := sTemp;
		END_IF
		
		//Info till sensorblock
		sensor7.bComError := FAULT;
		sensor7.rRawValue := AI7_PV;
		sensor7.sSensorConfig := AI7_PV1;
		
		//Ingång 8
		rTempArr[0] := wInputRegs1[15];
		rTempArr[1] := wInputRegs1[14];
		rTemp := fWordToReal(rTempArr);
		
		AI8_PV := fWordToReal(rTempArr);
				
		IF sensor8config.bResistance THEN
			
			AI8_PV1 := CONCAT('Givartyp: ', TO_STRING(sensor8config.sensorType));
		ELSE
			stemp := '0-10V';
			AI8_PV1 := sTemp;
		END_IF
		
		//Info till sensorblock
		sensor8.bComError := FAULT;
		sensor8.rRawValue := AI8_PV;
		sensor8.sSensorConfig := AI8_PV1;
		
		//Error 
		IF FB_MBReadInputRegs_Values.bError THEN
			FB_MBReadInputRegs_Values(bExecute := FALSE);
			iStep := 99;
		END_IF
	
		//Gå till nästa steg
		IF NOT FB_MBReadInputRegs_Values.bBusy AND NOT FB_MBReadInputRegs_Values.bError THEN
			FB_MBReadInputRegs_Values(bExecute := FALSE);
			bError := FALSE;
			iStep := 2;
		END_IF;
		
	2: 	//Läs config
		bBusy := TRUE;
		FB_MBReadRegs_Config.bExecute := TRUE;
	
		//Konfigurering
		wInputRegs2w[16] := config(sensor1config.bResistance,sensor1config.sensorType);
		wInputRegs2w[17] := config(sensor2config.bResistance,sensor2config.sensorType);
		wInputRegs2w[18] := config(sensor3config.bResistance,sensor3config.sensorType);
		wInputRegs2w[19] := config(sensor4config.bResistance,sensor4config.sensorType);
		wInputRegs2w[20] := config(sensor5config.bResistance,sensor5config.sensorType);
		wInputRegs2w[21] := config(sensor6config.bResistance,sensor6config.sensorType);
		wInputRegs2w[22] := config(sensor7config.bResistance,sensor7config.sensorType);
		wInputRegs2w[23] := config(sensor8config.bResistance,sensor8config.sensorType);
	
		FB_MBReadRegs_Config(
		sIPAddr:= modbusTCP.sIpAddr, 
		nTCPPort:= modbusTCP.nTCPPort, 
		nUnitID:= nUnitID, 
		nQuantity:= 8, 
		nMBAddr:= 16, 
		cbLength:= SIZEOF(wInputRegs2r), 
		pDestAddr:= ADR(wInputRegs2r), 
		bExecute:= , 
		tTimeout:= tTimeOut, 
		bBusy=> , 
		bError=> , 
		nErrId=> , 
		cbRead=> );

		//Error 
		IF FB_MBReadRegs_Config.bError THEN
			FB_MBReadRegs_Config(bExecute := FALSE);
			iStep := 99;
		END_IF
	
		//Next step
		IF NOT FB_MBReadRegs_Config.bBusy AND NOT FB_MBReadRegs_Config.bError THEN
			FB_MBReadRegs_Config(bExecute := FALSE);
		
			//Loop to check if config is different
			FOR arrIndex:=16 TO 23 BY 1 DO
				IF wInputRegs2r[arrIndex] = wInputRegs2w[arrIndex] THEN
			 		iConfigChanged := iConfigChanged;
				ELSE 
			 		iConfigChanged := iConfigChanged +1;
				END_IF
			END_FOR;
	
			IF iConfigChanged > 0 THEN
				bChangeConfig := TRUE;
				iStep := 3;
				bError := FALSE;
			ELSE 
				iStep := 4;
				bError := FALSE;
			END_IF
				
		END_IF;
	
	3: //Write if config is different from read value
		bBusy := TRUE;	
		IF bChangeConfig THEN
			FB_MBWriteRegs_Config.bExecute := TRUE;
		END_IF
			
		FB_MBWriteRegs_Config(
		sIPAddr:= modbusTCP.sIpAddr, 
		nTCPPort:= modbusTCP.nTCPPort, 
		nUnitID:= nUnitID, 
		nQuantity:= 8, 
		nMBAddr:= 16, 
		cbLength:= SIZEOF(wInputRegs2w), 
		pSrcAddr:= ADR(wInputRegs2w), 
		bExecute:=, 
		tTimeout:= tTimeOut, 
		bBusy=> , 
		bError=> , 
		nErrId=> );
		
		IF FB_MBWriteRegs_Config.bError THEN
			FB_MBWriteRegs_Config(bExecute := FALSE);
			iStep := 99;
		END_IF
	
		//Next step
		IF NOT FB_MBWriteRegs_Config.bBusy AND NOT FB_MBWriteRegs_Config.bError THEN
			FB_MBWriteRegs_Config(bExecute := FALSE);
			iConfigChanged := 0;
			bChangeConfig := FALSE; //Reset write
			bError := FALSE;
			iStep := 4;
		END_IF;
			
	4: //Done
		bBusy := FALSE;
		iStep := 0;

	99: //Error handling
		bBusy := FALSE;
		bError := TRUE;
		iStep := 0;
		
END_CASE
	
//Communication error
	fbKommTof(IN:=bError , PT:=T#20S , Q=> , ET=> );
	fbKommTon(bInput:=fbKommTof.Q , tAlarmDelay:=T#1M , bAutoReset:= , bAlarmOutput=> );
	FAULT :=fbKommTon.bAlarmOutput;
		
//Write busy	
	oaksgvl.aBModbusBusyFlagga[modbusTCP.iModbusLoop,nUnitID] := bBusy;

METHOD PRIVATE config : WORD
VAR_INPUT
	bResistance : BOOL; //0-10V (false) eller resistans (true)
	wSensorType : WORD;
	
END_VAR

VAR
	wOffset : WORD := 0; 
END_VAR
//Temperaturmätning
IF bResistance THEN

	wOffset := wSensorType;
	
	config.0 := FALSE; //Float
	config.1 := wOffset.0; 
	config.2 := wOffset.1; 
	config.3 := wOffset.2; 
	config.4 := wOffset.3;  
	config.5 := wOffset.4; 
	config.6 := wOffset.5; 
	config.7 := TRUE; //Välj resistans 
	config.8 := FALSE; 
	config.9 := FALSE; 
	config.10 := FALSE; 
	config.11 := FALSE; 
	config.12 := FALSE; 
	config.13 := FALSE; 
	config.14 := FALSE; 
	config.15 := FALSE; 
 
  
//Spänningsmätning
ELSE
	config.0 := FALSE; //Float
	config.1 := FALSE; 
	config.2 := FALSE; 
	config.3 := FALSE; 
	config.4 := FALSE;  
	config.5 := FALSE; 
	config.6 := FALSE; 
	config.7 := FALSE; //Välj resistans 
	config.8 := FALSE; 
	config.9 := FALSE; 
	config.10 := FALSE; 
	config.11 := FALSE; 
	config.12 := FALSE; 
	config.13 := FALSE; 
	config.14 := FALSE; 
	config.15 := FALSE; 
END_IF
END_METHOD

END_FUNCTION_BLOCK

// oaksModbusLibrary/Metz/fbMetzMR_AOP4
//Oaks AB
//2022-05-13 / Johan Bornemyr
//Funktionsblock för hantering av Metz MR IO-system. 
//MR-AOP4. Modul med 4 Analoga utgångar. Fysisk handställningsmöjlighet 0-10V på modul.
FUNCTION_BLOCK fbMetzMR_AOP4
VAR_INPUT
	bEnable : BOOL := TRUE; //Aktivering
	modbusTCP : ST_ModbusTCP;
	nUnitID: BYTE := 0;
	rAO1Setpoint : REAL := 0; //Börvärde Analog utgång 1 (0-100%)
	bAO1Invert : BOOL := FALSE; //Invertering utgång
	rAO1FallbackVoltage : REAL := 0; //Börvärde Analog utgång 1 (0-10V)
	rAO2Setpoint : REAL := 0; //Börvärde Analog utgång 2 (0-100%)
	bAO2Invert : BOOL := FALSE; //Invertering utgång
	rAO2FallbackVoltage : REAL := 0; //Börvärde Analog utgång 2 (0-10V)
	rAO3Setpoint : REAL := 0; //Börvärde Analog utgång 3 (0-100%)
	bAO3Invert : BOOL := FALSE; //Invertering utgång
	rAO3FallbackVoltage : REAL := 0; //Börvärde Analog utgång 3 (0-10V)
	rAO4Setpoint : REAL := 0; //Börvärde Analog utgång 4 (0-100%)
	bAO4Invert : BOOL := FALSE; //Invertering utgång
	rAO4FallbackVoltage : REAL := 0; //Börvärde Analog utgång 4 (0-10V)
END_VAR
	
VAR_INPUT PERSISTENT
	SP1 AT %M* : REAL := 0;//Komm.fels fördröjning IO~wp:[unit]ms[format]0.0
END_VAR

VAR_OUTPUT
	AO1_OP AT %M* : REAL;//Analog utgång 1~wp:[unit]V[format]0.00
	AO1_FAULT AT %M* : BOOL;//Omkopplare i fel läge utgång 1~wp:
	AO2_OP AT %M* : REAL;//Analog utgång 2~wp:[unit]V[format]0.00
	AO2_FAULT AT %M* : BOOL;//Omkopplare i fel läge utgång 2~wp:
	AO3_OP AT %M* : REAL;//Analog utgång 3~wp:[unit]V[format]0.00
	AO3_FAULT AT %M* : BOOL;//Omkopplare i fel läge utgång 3~wp:
	AO4_OP AT %M* : REAL;//Analog utgång 4~wp:[unit]V[format]0.00
	AO4_FAULT AT %M* : BOOL;//Omkopplare i fel läge utgång 4~wp:
	PV8 AT %M* : STRING;//Modbus konfiguering~wp:
	FAULT AT %M* : BOOL;//Kommunikationsfel~wp:
END_VAR
VAR
	tTimeOut : TIME :=T#5S;
	sIP: STRING(255);
	sPort: STRING(255);
	sModbusID: STRING(255);
	sModbusLoop: STRING(255);
	sTemp : STRING(255);	

	bSekvensFlagga : BOOL;
	iStep: INT;
	bError: BOOL;
	bBusy: BOOL;
	
	//Read output values and default values
	FB_MBReadRegs_ArrHolding1: FB_MBReadRegs;
	ArrHolding1 : ARRAY [0..7] OF WORD; //Holding

	//Outputs in manual mode
	FB_MBReadInputs_wDiscreteInputs: FB_MBReadInputs;
	wDiscreteInputs1 : WORD; //Discrete Input;
	
	fbAlarm_Output1man : fbAlarm;
	fbAlarm_Output2man : fbAlarm;
	fbAlarm_Output3man : fbAlarm;
	fbAlarm_Output4man : fbAlarm;

	//Communication error
	fbKommTof : tof; 
	fbKommTon : fbAlarm;
	
	fbReadWriteHoldingRegReal_ComError: fbReadWriteHoldingRegReal;
	
	//Configuration
	FB_MBWriteRegs_Config: FB_MBWriteRegs;
	wInputRegs2w : ARRAY[1..4] OF WORD; //Läs/skriv input regs modbus function 16.
	wInputRegs2r : ARRAY[1..4] OF WORD; //Läs/skriv input regs modbus function 16.
	iConfigChanged: INT;
	bChangeConfig: BOOL;
	arrIndex: INT;
	
	//Outputs
	FB_MBWriteRegs_Outputs: FB_MBWriteRegs;
	wInputRegsOutputsw : ARRAY[1..4] OF WORD; //Läs/skriv input regs modbus function 16.
		
	R_TRIG_Sekvens: R_TRIG;
END_VAR

//Sekvens	
	R_TRIG_Sekvens(CLK:= oaksGVL.aBModbusSekvens[modbusTCP.iModbusLoop] = BYTE_TO_INT(nUnitID), Q=> bSekvensFlagga);
	
	
//Modbus config
	sIP := CONCAT (modbusTCP.sIPAddr, '');
	sPort := CONCAT ('<br>Port: ', UINT_TO_STRING(modbusTCP.nTCPPort)); 								
	sModbusID := CONCAT('<br>ID: ', BYTE_TO_STRING(nUnitID));
	sModbusLoop := CONCAT('<br>Loop: ', INT_TO_STRING(modbusTCP.iModbusLoop));	

	sTemp := sIP;
	sTemp := CONCAT(sTemp, sPort);
	sTemp := CONCAT(sTemp, sModbusID);
	sTemp := CONCAT(sTemp, sModbusLoop);
	
	PV8 := sTemp;

	CASE iStep OF

	0: 	//Start/reset
		bBusy := FALSE;

		IF bEnable AND bSekvensFlagga THEN
			iStep := 1;
			bError := FALSE;
		END_IF
		
	1: 	//Read measured values
		bBusy := TRUE;
		
		FB_MBReadInputs_wDiscreteInputs.bExecute := TRUE;

		FB_MBReadInputs_wDiscreteInputs(
		sIPAddr:= modbusTCP.sIpAddr, 
		nTCPPort:= modbusTCP.nTCPPort, 
		nUnitID:= nUnitID, 
		nQuantity:= 4, 
		nMBAddr:= 0, 
		cbLength:= SIZEOF(wDiscreteInputs1), 
		pDestAddr:= ADR(wDiscreteInputs1),
		bExecute:=, 
		tTimeout:= tTimeOut, 
		bBusy=> , 
		bError=> , 
		nErrId=> , 
		cbRead=> );
	
		//Switch manual alarm
		fbAlarm_Output1man(bInput:= wDiscreteInputs1.0, tAlarmDelay:= T#3S, bAutoReset:= , bAlarmOutput=> AO1_FAULT);
		fbAlarm_Output2man(bInput:= wDiscreteInputs1.1, tAlarmDelay:= T#3S, bAutoReset:= , bAlarmOutput=> AO2_FAULT);
		fbAlarm_Output3man(bInput:= wDiscreteInputs1.2, tAlarmDelay:= T#3S, bAutoReset:= , bAlarmOutput=> AO3_FAULT);
		fbAlarm_Output4man(bInput:= wDiscreteInputs1.3, tAlarmDelay:= T#3S, bAutoReset:= , bAlarmOutput=> AO4_FAULT);
			
		//Error 
		IF FB_MBReadInputs_wDiscreteInputs.bError THEN
			FB_MBReadInputs_wDiscreteInputs(bExecute := FALSE);
			iStep := 99;
		END_IF
	
		//Next step
		IF NOT FB_MBReadInputs_wDiscreteInputs.bBusy AND NOT FB_MBReadInputs_wDiscreteInputs.bError THEN
			FB_MBReadInputs_wDiscreteInputs(bExecute := FALSE);
			bError := FALSE;
			iStep := 2;
		END_IF;
			
		
	2: //Read Data (Value on output)
		bBusy := TRUE;
		FB_MBReadRegs_ArrHolding1.bExecute := TRUE;

		//Read Holding 0-7
		FB_MBReadRegs_ArrHolding1(
		sIPAddr:= modbusTCP.sIpAddr, 
		nTCPPort:= modbusTCP.nTCPPort, 
		nUnitID:= nUnitID, 
		nQuantity:= 8, 
		nMBAddr:= 0, 
		cbLength:= SIZEOF(ArrHolding1), 
		pDestAddr:= ADR(ArrHolding1), 
		bExecute:=, 
		tTimeout:= tTimeOut, 
		bBusy=> ,
		bError=> , 
		nErrId=> , 
		cbRead=> );
	
		//Values
		AO1_OP := mRawToAnalog(ArrHolding1[0]); //0
		AO2_OP := mRawToAnalog(ArrHolding1[1]); //1
		AO3_OP := mRawToAnalog(ArrHolding1[2]); //2
		AO4_OP := mRawToAnalog(ArrHolding1[3]); //3

		//Error 
		IF FB_MBReadRegs_ArrHolding1.bError THEN
			FB_MBReadRegs_ArrHolding1(bExecute := FALSE);
			iStep := 99;
		END_IF
	
		//Gå till nästa steg
		IF NOT FB_MBReadRegs_ArrHolding1.bBusy AND NOT FB_MBReadRegs_ArrHolding1.bError THEN
			FB_MBReadRegs_ArrHolding1(bExecute := FALSE);
			bError := FALSE;
			iStep := 3;
		END_IF;

	3: //Read/Write communication error timedelay (config)
		bBusy := TRUE;

		//User input
		IF SP1 < 0 THEN
			SP1 := 0;
		END_IF;
		
		IF SP1 > 65535 THEN
			SP1 := 655;
		END_IF;
		
		fbReadWriteHoldingRegReal_ComError.bEnable := TRUE;
		
		fbReadWriteHoldingRegReal_ComError(
		sIPAddr:= modbusTCP.sIpAddr, 
		nTCPPort:= modbusTCP.nTCPPort, 
		nUnitID:= nUnitID, 
		mBusAdr:= 66, 
		bEnable:= , 
		tTimeout:= tTimeOut, 
		rReal:= SP1, 
		uiFaktor:= 100, 
		bError=> , 
		bBusy=> , 
		bSuccess=> );
				
		//Error 
		IF fbReadWriteHoldingRegReal_ComError.bError THEN
			fbReadWriteHoldingRegReal_ComError(bEnable := FALSE);
			iStep := 99;
		END_IF
	
		//Gå till nästa steg
		IF NOT fbReadWriteHoldingRegReal_ComError.bBusy AND NOT fbReadWriteHoldingRegReal_ComError.bError THEN
			fbReadWriteHoldingRegReal_ComError(bEnable := FALSE);
			bError := FALSE;
			iStep := 4;
		END_IF;

	4:	//Read/Write default values (config)
		
		//Config in IO
		wInputRegs2r[1] := ArrHolding1[4]; //4;
		wInputRegs2r[2] := ArrHolding1[5]; //5;
		wInputRegs2r[3] := ArrHolding1[6]; //6;
		wInputRegs2r[4] := ArrHolding1[7]; //7;
		//Config in PLC	
		wInputRegs2w[1] := mAnalogToRawFallback(rAO1FallbackVoltage); //4;
		wInputRegs2w[2] := mAnalogToRawFallback(rAO2FallbackVoltage); //5;
		wInputRegs2w[3] := mAnalogToRawFallback(rAO3FallbackVoltage); //6;
		wInputRegs2w[4] := mAnalogToRawFallback(rAO4FallbackVoltage); //7;
		
		FOR arrIndex:=1 TO 4 BY 1 DO
				IF wInputRegs2r[arrIndex] = wInputRegs2w[arrIndex] THEN
			 		iConfigChanged := iConfigChanged;
				ELSE 
			 		iConfigChanged := iConfigChanged +1;
				END_IF
		END_FOR;
	
		IF iConfigChanged > 0 THEN
			bChangeConfig := TRUE;
			iStep := 5;
			bError := FALSE;
		ELSE 
			iStep := 6;
			bError := FALSE;
		END_IF
 
	5: //Write if config is different from read value
		bBusy := TRUE;	
		IF bChangeConfig THEN
			FB_MBWriteRegs_Config.bExecute := TRUE;
		END_IF
			
		FB_MBWriteRegs_Config(
		sIPAddr:= modbusTCP.sIpAddr, 
		nTCPPort:= modbusTCP.nTCPPort, 
		nUnitID:= nUnitID, 
		nQuantity:= 4, 
		nMBAddr:= 4, 
		cbLength:= SIZEOF(wInputRegs2w), 
		pSrcAddr:= ADR(wInputRegs2w), 
		bExecute:=, 
		tTimeout:= tTimeOut, 
		bBusy=> , 
		bError=> , 
		nErrId=> );
		
		IF FB_MBWriteRegs_Config.bError THEN
			FB_MBWriteRegs_Config(bExecute := FALSE);
			iStep := 99;
		END_IF
	
		//Next step
		IF NOT FB_MBWriteRegs_Config.bBusy AND NOT FB_MBWriteRegs_Config.bError THEN
			FB_MBWriteRegs_Config(bExecute := FALSE);
			iConfigChanged := 0;
			bChangeConfig := FALSE; //Reset write
			bError := FALSE;
			iStep := 6;
		END_IF;

	6: //Write outputs
		bBusy := TRUE;	
			
		wInputRegsOutputsw[1] := mAnalogToRaw(rAO1Setpoint,bAO1Invert);
		wInputRegsOutputsw[2] := mAnalogToRaw(rAO2Setpoint,bAO2Invert);
		wInputRegsOutputsw[3] := mAnalogToRaw(rAO3Setpoint,bAO3Invert);
		wInputRegsOutputsw[4] := mAnalogToRaw(rAO4Setpoint,bAO4Invert);
		
		FB_MBWriteRegs_Outputs.bExecute := TRUE;
		
		FB_MBWriteRegs_Outputs(
		sIPAddr:= modbusTCP.sIpAddr, 
		nTCPPort:= modbusTCP.nTCPPort, 
		nUnitID:= nUnitID, 
		nQuantity:= 4, 
		nMBAddr:= 0, 
		cbLength:= SIZEOF(wInputRegsOutputsw), 
		pSrcAddr:= ADR(wInputRegsOutputsw), 
		bExecute:=, 
		tTimeout:= tTimeOut, 
		bBusy=> , 
		bError=> , 
		nErrId=> );
		
		IF FB_MBWriteRegs_Outputs.bError THEN
			FB_MBWriteRegs_Outputs(bExecute := FALSE);
			iStep := 99;
		END_IF
	
		//Next step
		IF NOT FB_MBWriteRegs_Outputs.bBusy AND NOT FB_MBWriteRegs_Outputs.bError THEN
			FB_MBWriteRegs_Outputs(bExecute := FALSE);
			bError := FALSE;
			iStep := 20;
		END_IF;

	20: //Done
		bBusy := FALSE;
		iStep := 0;

	99: //Error handling
		bBusy := FALSE;
		bError := TRUE;
		iStep := 0;
		
END_CASE

//Communication error
	fbKommTof(IN:=bError , PT:=T#20S , Q=> , ET=> );
	fbKommTon(bInput:=fbKommTof.Q , tAlarmDelay:=T#1M , bAutoReset:= , bAlarmOutput=> );
	FAULT :=fbKommTon.bAlarmOutput;
		
//Write busy	
	oaksgvl.aBModbusBusyFlagga[modbusTCP.iModbusLoop,nUnitID] := bBusy;

METHOD mAnalogToRaw : WORD
VAR_INPUT
	rValueToConvert : REAL; //Rå-värde
	bAOInvert : BOOL := FALSE; //Invertering utgång
END_VAR

VAR
	x1 : REAL;
	x2 : REAL;
	y1 : REAL;
	y2 : REAL;
	rPercent : REAL;
	rRawAnalog : REAL;
	rInternalVal: REAL;
END_VAR
//0-100%
rInternalVal := LIMIT(0,rValueToConvert,100);

x1 := 0; 
x2 := 100; 
y1 := 0; 
y2 := 10;
rPercent := fScale2p(rInternalVal,y1, y2, x1, x2);

//0-10V
x1 := 0; 
x2 := 10.24; 
y1 := 0; 
y2 := 32767;
IF NOT bAOInvert THEN
	rRawAnalog := fScale2p(rPercent, y1, y2, x1, x2);
ELSE
	rRawAnalog := fScale2p(rPercent, y2, y1, x1, x2);	
END_IF
mAnalogToRaw := fRealtoWord(rRawAnalog, 1);
END_METHOD

METHOD mAnalogToRawFallback : WORD
VAR_INPUT
	rValueToConvert : REAL; //Rå-värde
END_VAR

VAR
	x1 : REAL;
	x2 : REAL;
	y1 : REAL;
	y2 : REAL;
	rPercent : REAL;
	rRawAnalog : REAL;
	rInternalVal: REAL;
END_VAR
//0-100%
rInternalVal := LIMIT(0,rValueToConvert,100);

x1 := 0; 
x2 := 100; 
y1 := 0; 
y2 := 10;
rPercent := fScale2p(rInternalVal,y1, y2, x1, x2);

//0-10V
x1 := 0; 
x2 := 10.24; 
y1 := 0; 
y2 := 32767;

mAnalogToRawFallback := fRealtoWord(fScale2p(rPercent, y1, y2, x1, x2), 1);
END_METHOD

METHOD mRawToAnalog : REAL
VAR_INPUT
	rValueToConvert : WORD; //Rå-värde
END_VAR

VAR
	x1 : REAL;
	x2 : REAL;
	y1 : REAL;
	y2 : REAL;
	rTemp : REAL;
END_VAR
//0-10V
rTemp := fSignedConverter(rValueToConvert);

x1 := 0; 
x2 := 32767;
y1 := 0; 
y2 := 10.24; 
mRawToAnalog := fScale2p(rTemp, y1, y2, x1, x2);
END_METHOD

END_FUNCTION_BLOCK

// oaksModbusLibrary/Metz/fbMetzMR_DI10
//Oaks AB
//2022-05-13 / Johan Bornemyr
//Funktionsblock för hantering av Metz MR IO-system. 
//MR-DI10. Modul med 10 Digitala ingångar.
FUNCTION_BLOCK fbMetzMR_DI10
VAR_INPUT
	bEnable : BOOL := TRUE; //Aktivering
	modbusTCP : ST_ModbusTCP;
	nUnitID: BYTE := 0;
END_VAR
VAR_OUTPUT
	
	DI1_V AT %M* : BOOL;//Digital ingång 1~wp:[trendoptions]i:14400, t:1
	DI2_V AT %M* : BOOL;//Digital ingång 2~wp:[trendoptions]i:14400, t:1
	DI3_V AT %M* : BOOL;//Digital ingång 3~wp:[trendoptions]i:14400, t:1
	DI4_V AT %M* : BOOL;//Digital ingång 4~wp:[trendoptions]i:14400, t:1
	DI5_V AT %M* : BOOL;//Digital ingång 5~wp:[trendoptions]i:14400, t:1
	DI6_V AT %M* : BOOL;//Digital ingång 6~wp:[trendoptions]i:14400, t:1
	DI7_V AT %M* : BOOL;//Digital ingång 7~wp:[trendoptions]i:14400, t:1
	DI8_V AT %M* : BOOL;//Digital ingång 8~wp:[trendoptions]i:14400, t:1
	DI9_V AT %M* : BOOL;//Digital ingång 9~wp:[trendoptions]i:14400, t:1
	DI10_V AT %M* : BOOL;//Digital ingång 10~wp:[trendoptions]i:14400, t:1

	
	PV8 AT %M* : STRING;//Modbus konfiguering~wp:
	FAULT AT %M* : BOOL;//Kommunikationsfel~wp:
	
END_VAR
VAR
	tTimeOut : TIME :=T#5S;
	sIP: STRING(255);
	sPort: STRING(255);
	sModbusID: STRING(255);
	sModbusLoop: STRING(255);
	sTemp : STRING(255);
	bSekvensFlagga : BOOL;
		
	FB_MBReadRegs_InputRegs1: FB_MBReadInputRegs;
	wInputRegs1 : WORD; //Read input regs modbus function 4. 
		
	//Communication error
	fbKommTof : tof; 
	fbKommTon : fbAlarm;

	
	R_TRIG_Sekvens: R_TRIG;
END_VAR

//Sekvens	
	R_TRIG_Sekvens(CLK:= oaksGVL.aBModbusSekvens[modbusTCP.iModbusLoop] = BYTE_TO_INT(nUnitID), Q=> bSekvensFlagga);
	
//Modbus config
	sIP := CONCAT (modbusTCP.sIPAddr, '');
	sPort := CONCAT ('<br>Port: ', UINT_TO_STRING(modbusTCP.nTCPPort)); 								
	sModbusID := CONCAT('<br>ID: ', BYTE_TO_STRING(nUnitID));
	sModbusLoop := CONCAT('<br>Loop: ', INT_TO_STRING(modbusTCP.iModbusLoop));	

	sTemp := sIP;
	sTemp := CONCAT(sTemp, sPort);
	sTemp := CONCAT(sTemp, sModbusID);
	sTemp := CONCAT(sTemp, sModbusLoop);
	
	PV8 := sTemp;
	
	//Read Input states
	FB_MBReadRegs_InputRegs1(
	sIPAddr:= modbusTCP.sIpAddr, 
	nTCPPort:= modbusTCP.nTCPPort, 
	nUnitID:= nUnitID, 
	nQuantity:= 1, 
	nMBAddr:= 0, 
	cbLength:= SIZEOF(wInputRegs1), 
	pDestAddr:= ADR(wInputRegs1), 
	bExecute:= bSekvensFlagga AND bEnable, 
	tTimeout:= tTimeOut, 
	bBusy=> , 
	bError=> , 
	nErrId=> , 
	cbRead=> );
	
	DI1_V := wInputRegs1.0;
	DI2_V := wInputRegs1.1;
	DI3_V := wInputRegs1.2;
	DI4_V := wInputRegs1.3;
	DI5_V := wInputRegs1.4;
	DI6_V := wInputRegs1.5;
	DI7_V := wInputRegs1.6;
	DI8_V := wInputRegs1.7;
	DI9_V := wInputRegs1.8;
	DI10_V := wInputRegs1.9;
		
//Communication error
	fbKommTof(IN:=FB_MBReadRegs_InputRegs1.bError , PT:=T#20S , Q=> , ET=> );
	fbKommTon(bInput:=fbKommTof.Q , tAlarmDelay:=T#1M , bAutoReset:= , bAlarmOutput=> );
	FAULT :=fbKommTon.bAlarmOutput;
		
//Write busy	
	oaksgvl.aBModbusBusyFlagga[modbusTCP.iModbusLoop,nUnitID] := FB_MBReadRegs_InputRegs1.bBusy;

END_FUNCTION_BLOCK

// oaksModbusLibrary/Metz/fbMetzMR_DI4
//Oaks AB
//2022-05-13 / Johan Bornemyr
//Funktionsblock för hantering av Metz MR IO-system. 
//MR-DI4. Modul med 4 Digitala ingångar. För att avläsa potentialfria växlings lägen.
FUNCTION_BLOCK fbMetzMR_DI4
VAR_INPUT
	bEnable : BOOL := TRUE; //Aktivering
	modbusTCP : ST_ModbusTCP;
	nUnitID: BYTE := 0;
END_VAR
VAR_OUTPUT
	
	DI1_V AT %M* : BOOL;//Digital ingång 1~wp:[trendoptions]i:14400, t:1
	DI2_V AT %M* : BOOL;//Digital ingång 2~wp:[trendoptions]i:14400, t:1
	DI3_V AT %M* : BOOL;//Digital ingång 3~wp:[trendoptions]i:14400, t:1
	DI4_V AT %M* : BOOL;//Digital ingång 4~wp:[trendoptions]i:14400, t:1
	
	PV8 AT %M* : STRING;//Modbus konfiguering~wp:
	FAULT AT %M* : BOOL;//Kommunikationsfel~wp:
	
END_VAR
VAR
	tTimeOut : TIME :=T#5S;
	sIP: STRING(255);
	sPort: STRING(255);
	sModbusID: STRING(255);
	sModbusLoop: STRING(255);
	sTemp : STRING(255);
	bSekvensFlagga : BOOL;
		
	FB_MBReadRegs_InputRegs1: FB_MBReadInputRegs;
	wInputRegs1 : WORD; //Read input regs modbus function 4. 
		
	//Communication error
	fbKommTof : tof; 
	fbKommTon : fbAlarm;
	
	R_TRIG_Sekvens: R_TRIG;
END_VAR

//Sekvens	
	R_TRIG_Sekvens(CLK:= oaksGVL.aBModbusSekvens[modbusTCP.iModbusLoop] = BYTE_TO_INT(nUnitID), Q=> bSekvensFlagga);
	
//Modbus config
	sIP := CONCAT (modbusTCP.sIPAddr, '');
	sPort := CONCAT ('<br>Port: ', UINT_TO_STRING(modbusTCP.nTCPPort)); 								
	sModbusID := CONCAT('<br>ID: ', BYTE_TO_STRING(nUnitID));
	sModbusLoop := CONCAT('<br>Loop: ', INT_TO_STRING(modbusTCP.iModbusLoop));	

	sTemp := sIP;
	sTemp := CONCAT(sTemp, sPort);
	sTemp := CONCAT(sTemp, sModbusID);
	sTemp := CONCAT(sTemp, sModbusLoop);
	
	PV8 := sTemp;
	
	//Read Input states
	FB_MBReadRegs_InputRegs1(
	sIPAddr:= modbusTCP.sIpAddr, 
	nTCPPort:= modbusTCP.nTCPPort, 
	nUnitID:= nUnitID, 
	nQuantity:= 1, 
	nMBAddr:= 0, 
	cbLength:= SIZEOF(wInputRegs1), 
	pDestAddr:= ADR(wInputRegs1), 
	bExecute:= bSekvensFlagga AND bEnable, 
	tTimeout:= tTimeOut, 
	bBusy=> , 
	bError=> , 
	nErrId=> , 
	cbRead=> );
	
	DI1_V := wInputRegs1.0;
	DI2_V := wInputRegs1.1;
	DI3_V := wInputRegs1.2;
	DI4_V := wInputRegs1.3;
			
//Communication error
	fbKommTof(IN:=FB_MBReadRegs_InputRegs1.bError , PT:=T#20S , Q=> , ET=> );
	fbKommTon(bInput:=fbKommTof.Q , tAlarmDelay:=T#1M , bAutoReset:= , bAlarmOutput=> );
	FAULT :=fbKommTon.bAlarmOutput;
		
//Write busy	
	oaksgvl.aBModbusBusyFlagga[modbusTCP.iModbusLoop,nUnitID] := FB_MBReadRegs_InputRegs1.bBusy;

END_FUNCTION_BLOCK

// oaksModbusLibrary/Metz/fbMetzMR_DO4
//Oaks AB
//2022-05-13 / Johan Bornemyr
//Funktionsblock för hantering av Metz MR IO-system. 
//MR-AOP4. Modul med 4 digitala utgångar. Fysisk handställningsmöjlighet av/på på modul.
FUNCTION_BLOCK fbMetzMR_DO4
VAR_INPUT
	bEnable : BOOL := TRUE; //Aktivering
	modbusTCP : ST_ModbusTCP;
	nUnitID: BYTE := 0;
	bDO1 : BOOL := FALSE; //Manöver digital utgång 1
	bDO1fallback : BOOL; //Värde vid komm.fel utgång 1
	bDO2 : BOOL := FALSE; //Manöver digital utgång 2
	bDO2fallback : BOOL; //Värde vid komm.fel utgång 2
	bDO3 : BOOL := FALSE; //Manöver digital utgång 3
	bDO3fallback : BOOL; //Värde vid komm.fel utgång 3
	bDO4 : BOOL := FALSE; //Manöver digital utgång 4
	bDO4fallback : BOOL; //Värde vid komm.fel utgång 4
END_VAR
	
VAR_INPUT PERSISTENT
	SP1 AT %M* : REAL := 0;//Komm.fels fördröjning IO~wp:[unit]ms[format]0.0
END_VAR

VAR_OUTPUT
	DO1_V AT %M* : BOOL :=FALSE;//Digital utgång 1~wp:
	DO1_FAULT AT %M* : BOOL :=FALSE;//Omkopplare i fel läge utgång 1~wp:
	DO2_V AT %M* : BOOL :=FALSE;//Digital utgång 2~wp:
	DO2_FAULT AT %M* : BOOL :=FALSE;//Omkopplare i fel läge utgång 2~wp:
	DO3_V AT %M* : BOOL :=FALSE;//Digital utgång 3~wp:
	DO3_FAULT AT %M* : BOOL :=FALSE;//Omkopplare i fel läge utgång 3~wp:
	DO4_V AT %M* : BOOL :=FALSE;//Digital utgång 4~wp:
	DO4_FAULT AT %M* : BOOL :=FALSE;//Omkopplare i fel läge utgång 4~wp:
	
	PV8 AT %M* : STRING;//Modbus konfiguering~wp:
	FAULT AT %M* : BOOL;//Kommunikationsfel~wp:
END_VAR
VAR
	tTimeOut : TIME :=T#5S;
	sIP: STRING(255);
	sPort: STRING(255);
	sModbusID: STRING(255);
	sModbusLoop: STRING(255);
	sTemp : STRING(255);	

	bSekvensFlagga : BOOL;
	iStep: INT;
	bError: BOOL;
	bBusy: BOOL;
	
	//Read output values and default values
	FB_MBReadRegs_ArrHolding1: FB_MBReadRegs;
	ArrHolding1 : ARRAY [0..7] OF WORD; //Holding

	fbAlarm_Output1man : fbAlarm;
	fbAlarm_Output2man : fbAlarm;
	fbAlarm_Output3man : fbAlarm;
	fbAlarm_Output4man : fbAlarm;

	//Communication error
	fbKommTof : tof; 
	fbKommTon : fbAlarm;
	fbReadWriteHoldingRegReal_ComError: fbReadWriteHoldingRegReal;
	
	//Configuration
	FB_MBWriteRegs_Config: FB_MBWriteSingleReg;
	wWriteConfig : WORD; //Läs/skriv input regs modbus function 4.
	wReadConfig : WORD; //Läs/skriv input regs modbus function 4.
		
	//Outputs
	FB_MBWriteRegs_Outputs: FB_MBWriteSingleReg;
	wWriteOutputs : WORD; //Läs/skriv input regs modbus function 6.
		
	R_TRIG_Sekvens: R_TRIG;
END_VAR

//Sekvens
	R_TRIG_Sekvens(CLK:= oaksGVL.aBModbusSekvens[modbusTCP.iModbusLoop] = BYTE_TO_INT(nUnitID), Q=> bSekvensFlagga);
	
//Modbus config
	sIP := CONCAT (modbusTCP.sIPAddr, '');
	sPort := CONCAT ('<br>Port: ', UINT_TO_STRING(modbusTCP.nTCPPort)); 								
	sModbusID := CONCAT('<br>ID: ', BYTE_TO_STRING(nUnitID));
	sModbusLoop := CONCAT('<br>Loop: ', INT_TO_STRING(modbusTCP.iModbusLoop));	

	sTemp := sIP;
	sTemp := CONCAT(sTemp, sPort);
	sTemp := CONCAT(sTemp, sModbusID);
	sTemp := CONCAT(sTemp, sModbusLoop);
	
	PV8 := sTemp;

	CASE iStep OF

	0: 	//Start/reset
		bBusy := FALSE;
						
		IF bEnable AND bSekvensFlagga THEN
			iStep := 1;
			bError := FALSE;
		END_IF
		
	1: //Read Data (Value on output)
		bBusy := TRUE;
		FB_MBReadRegs_ArrHolding1.bExecute := TRUE;

		//Read Values
		FB_MBReadRegs_ArrHolding1(
			sIPAddr:= modbusTCP.sIpAddr, 
			nTCPPort:= modbusTCP.nTCPPort, 
			nUnitID:= nUnitID, 
			nQuantity:= 2, 
			nMBAddr:= 0, 
			cbLength:= SIZEOF(ArrHolding1), 
			pDestAddr:= ADR(ArrHolding1), 
			bExecute:=, 
			tTimeout:= tTimeOut, 
			bBusy=> ,
			bError=> , 
			nErrId=> , 
			cbRead=> );
	
		//Values
		DO1_V := ArrHolding1[0].0;
		DO2_V := ArrHolding1[0].1;
		DO3_V := ArrHolding1[0].2;
		DO4_V := ArrHolding1[0].3;
		
		//Switch manual alarm
		fbAlarm_Output1man(bInput:= ArrHolding1[0].4, tAlarmDelay:= T#3S, bAutoReset:= , bAlarmOutput=> DO1_FAULT);
		fbAlarm_Output2man(bInput:= ArrHolding1[0].5, tAlarmDelay:= T#3S, bAutoReset:= , bAlarmOutput=> DO2_FAULT);
		fbAlarm_Output3man(bInput:= ArrHolding1[0].6, tAlarmDelay:= T#3S, bAutoReset:= , bAlarmOutput=> DO3_FAULT);
		fbAlarm_Output4man(bInput:= ArrHolding1[0].7, tAlarmDelay:= T#3S, bAutoReset:= , bAlarmOutput=> DO4_FAULT);

		//Error 
		IF FB_MBReadRegs_ArrHolding1.bError THEN
			FB_MBReadRegs_ArrHolding1(bExecute := FALSE);
			iStep := 99;
		END_IF
	
		//Gå till nästa steg
		IF NOT FB_MBReadRegs_ArrHolding1.bBusy AND NOT FB_MBReadRegs_ArrHolding1.bError THEN
			FB_MBReadRegs_ArrHolding1(bExecute := FALSE);
			bError := FALSE;
			iStep := 2;
		END_IF;

	2: //Read/Write communication error timedelay (config)
		bBusy := TRUE;

		//User input
		IF SP1 < 0 THEN
			SP1 := 0;
		END_IF;
		
		IF SP1 > 65535 THEN
			SP1 := 655;
		END_IF;
		
		fbReadWriteHoldingRegReal_ComError.bEnable := TRUE;
		
		fbReadWriteHoldingRegReal_ComError(
			sIPAddr:= modbusTCP.sIpAddr, 
			nTCPPort:= modbusTCP.nTCPPort, 
			nUnitID:= nUnitID, 
			mBusAdr:= 66, 
			bEnable:= , 
			tTimeout:= tTimeOut, 
			rReal:= SP1, 
			uiFaktor:= 100, 
			bError=> , 
			bBusy=> , 
			bSuccess=> );
				
		//Error 
		IF fbReadWriteHoldingRegReal_ComError.bError THEN
			fbReadWriteHoldingRegReal_ComError(bEnable := FALSE);
			iStep := 99;
		END_IF
	
		//Gå till nästa steg
		IF NOT fbReadWriteHoldingRegReal_ComError.bBusy AND NOT fbReadWriteHoldingRegReal_ComError.bError THEN
			fbReadWriteHoldingRegReal_ComError(bEnable := FALSE);
			bError := FALSE;
			iStep := 3;
		END_IF;
	
	3:	//Read/Write default values (config)
		//Config in IO
		wReadConfig.0 := ArrHolding1[1].0;
		wReadConfig.1 := ArrHolding1[1].1;
		wReadConfig.2 := ArrHolding1[1].2;
		wReadConfig.3 := ArrHolding1[1].3;
		//Config in PLC	
		wWriteConfig.0 := bDO1fallback; 
		wWriteConfig.1 := bDO2fallback;
		wWriteConfig.2 := bDO3fallback;
		wWriteConfig.3 := bDO4fallback;
		
		bBusy := TRUE;	
		IF wReadConfig <> wWriteConfig THEN
			FB_MBWriteRegs_Config.bExecute := TRUE;
		END_IF
		
		FB_MBWriteRegs_Config(
			sIPAddr:= modbusTCP.sIpAddr, 
			nTCPPort:= modbusTCP.nTCPPort, 
			nUnitID:= nUnitID,
			nMBAddr:= 1,
			nValue:= wWriteConfig, 
			bExecute:= , 
			tTimeout:= tTimeout , 
			bBusy=> , 
			bError=> , 
			nErrId=> );
			
		IF FB_MBWriteRegs_Config.bError THEN
			FB_MBWriteRegs_Config(bExecute := FALSE);
			iStep := 99;
		END_IF
	
		//Next step
		IF NOT FB_MBWriteRegs_Config.bBusy AND NOT FB_MBWriteRegs_Config.bError THEN
			FB_MBWriteRegs_Config(bExecute := FALSE);
			bError := FALSE;
			iStep := 4;
		END_IF;

	4: //Write outputs
		bBusy := TRUE;	
			
		wWriteOutputs.0 := bDO1;
		wWriteOutputs.1 := bDO2;
		wWriteOutputs.2 := bDO3;
		wWriteOutputs.3 := bDO4;
		
		FB_MBWriteRegs_Outputs.bExecute := TRUE;
		
		FB_MBWriteRegs_Outputs(
			sIPAddr:= modbusTCP.sIpAddr, 
			nTCPPort:= modbusTCP.nTCPPort, 
			nUnitID:= nUnitID,
			nMBAddr:= 0,
			nValue:= wWriteOutputs, 
			bExecute:= , 
			tTimeout:= tTimeout , 
			bBusy=> , 
			bError=> , 
			nErrId=> );
				
		IF FB_MBWriteRegs_Outputs.bError THEN
			FB_MBWriteRegs_Outputs(bExecute := FALSE);
			iStep := 99;
		END_IF
	
		//Next step
		IF NOT FB_MBWriteRegs_Outputs.bBusy AND NOT FB_MBWriteRegs_Outputs.bError THEN
			FB_MBWriteRegs_Outputs(bExecute := FALSE);
			bError := FALSE;
			iStep := 20;
		END_IF;

	20: //Done
		bBusy := FALSE;
		iStep := 0;
		

	99: //Error handling
		bBusy := FALSE;
		bError := TRUE;
		iStep := 0;
		
END_CASE

